(* PLC project Untitled1, Eindhoven University of Technology (TU/e) CIF to Structured Text 0.0 *)
(* stored: creationDateTime 1970-01-01T01:00:00 *)

TYPE STATE : STRUCT
  curTime : LREAL;
  dvar_M_HPC1_HWPump1_ON AT %Q* : BOOL;
  dvar_M_HPC1_HWPump1 AT %Q* : enum_E;
  dvar_M_HPC1_HWPump2_ON AT %Q* : BOOL;
  dvar_M_HPC1_HWPump2 AT %Q* : enum_E;
  dvar_M_HPC1_HWSensorS1 AT %Q* : enum_E;
  dvar_M_HPC1_HWSensorS2 AT %Q* : enum_E;
  dvar_M_HPC1_HWSensorS3 AT %Q* : enum_E;
  dvar_M_HPC1_HWSensorS4 AT %Q* : enum_E;
  dvar_M_HPC1_HWSensorS5 AT %Q* : enum_E;
  dvar_M_HWHPC1ControlButtonAuto_StopLoop AT %Q* : BOOL;
  dvar_M_HWHPC1ControlButtonAuto AT %Q* : enum_E;
  dvar_M_HWHPC1ControlButtonManual_StopLoop AT %Q* : BOOL;
  dvar_M_HWHPC1ControlButtonManual AT %Q* : enum_E;
  dvar_M_HWHPC1ControlMode_AUTO AT %Q* : BOOL;
  dvar_M_HWHPC1ControlMode AT %Q* : enum_E;
  dvar_M_HWHPC1Mode_DRAIN AT %Q* : BOOL;
  dvar_M_HWHPC1Mode_STORE AT %Q* : BOOL;
  dvar_M_HWHPC1Mode_OFF AT %Q* : BOOL;
  dvar_M_HWHPC1Mode AT %Q* : enum_E;
  dvar_M_HWHPC1ModeButtonDrain_StopLoop AT %Q* : BOOL;
  dvar_M_HWHPC1ModeButtonDrain AT %Q* : enum_E;
  dvar_M_HWHPC1ModeButtonOff_StopLoop AT %Q* : BOOL;
  dvar_M_HWHPC1ModeButtonOff AT %Q* : enum_E;
  dvar_M_HWHPC1ModeButtonStore_StopLoop AT %Q* : BOOL;
  dvar_M_HWHPC1ModeButtonStore AT %Q* : enum_E;
  dvar_M_HWModeTraffictube1Observer AT %Q* : enum_E;
  dvar_M_HWModeTraffictube2Observer AT %Q* : enum_E;
  dvar_M_HWMPCControlButtonAuto_StopLoop AT %Q* : BOOL;
  dvar_M_HWMPCControlButtonAuto AT %Q* : enum_E;
  dvar_M_HWMPCControlButtonManual_StopLoop AT %Q* : BOOL;
  dvar_M_HWMPCControlButtonManual AT %Q* : enum_E;
  dvar_M_HWMPCControlMode_AUTO AT %Q* : BOOL;
  dvar_M_HWMPCControlMode AT %Q* : enum_E;
  dvar_M_HWMPCMode_DRAIN AT %Q* : BOOL;
  dvar_M_HWMPCMode_STORE AT %Q* : BOOL;
  dvar_M_HWMPCMode_OFF AT %Q* : BOOL;
  dvar_M_HWMPCMode AT %Q* : enum_E;
  dvar_M_HWMPCModeButtonDrain_StopLoop AT %Q* : BOOL;
  dvar_M_HWMPCModeButtonDrain AT %Q* : enum_E;
  dvar_M_HWMPCModeButtonOff_StopLoop AT %Q* : BOOL;
  dvar_M_HWMPCModeButtonOff AT %Q* : enum_E;
  dvar_M_HWMPCModeButtonStore_StopLoop AT %Q* : BOOL;
  dvar_M_HWMPCModeButtonStore AT %Q* : enum_E;
  dvar_M_HWMutex1_Here AT %Q* : BOOL;
  dvar_M_HWMutex1_SendingAway AT %Q* : BOOL;
  dvar_M_HWMutex1 AT %Q* : enum_E;
  dvar_M_HWMutex2_Here AT %Q* : BOOL;
  dvar_M_HWMutex2_SendingAway AT %Q* : BOOL;
  dvar_M_HWMutex2 AT %Q* : enum_E;
  dvar_M_HWMutex3_Here AT %Q* : BOOL;
  dvar_M_HWMutex3_SendingAway AT %Q* : BOOL;
  dvar_M_HWMutex3 AT %Q* : enum_E;
  dvar_M_HWMutex4_Here AT %Q* : BOOL;
  dvar_M_HWMutex4_SendingAway AT %Q* : BOOL;
  dvar_M_HWMutex4 AT %Q* : enum_E;
  dvar_M_MPC_HWPomprichting_HPC1 AT %Q* : BOOL;
  dvar_M_MPC_HWPomprichting AT %Q* : enum_E;
  dvar_M_MPC_HWPump1_ON AT %Q* : BOOL;
  dvar_M_MPC_HWPump1 AT %Q* : enum_E;
  dvar_M_MPC_HWPump2_ON AT %Q* : BOOL;
  dvar_M_MPC_HWPump2 AT %Q* : enum_E;
  dvar_M_MPC_HWSensorS1 AT %Q* : enum_E;
  dvar_M_MPC_HWSensorS2 AT %Q* : enum_E;
  dvar_M_MPC_HWSensorS3 AT %Q* : enum_E;
  dvar_M_MPC_HWSensorS4 AT %Q* : enum_E;
  dvar_M_MPC_HWSensorS5 AT %Q* : enum_E;
  dvar_M_Mutex1Home_TokenTracker AT %Q* : enum_E;
  dvar_M_Mutex2Home_TokenTracker AT %Q* : enum_E;
  dvar_M_Mutex3Home_TokenTracker AT %Q* : enum_E;
  dvar_M_Mutex4Home_TokenTracker AT %Q* : enum_E;
  dvar_M_Pumpcellars_HeadPumpcellar1_Control_ButtonAuto AT %Q* : enum_E;
  dvar_M_Pumpcellars_HeadPumpcellar1_Control_ButtonDrain AT %Q* : enum_E;
  dvar_M_Pumpcellars_HeadPumpcellar1_Control_ButtonManual AT %Q* : enum_E;
  dvar_M_Pumpcellars_HeadPumpcellar1_Control_ButtonOff AT %Q* : enum_E;
  dvar_M_Pumpcellars_HeadPumpcellar1_Control_ButtonStore AT %Q* : enum_E;
  dvar_M_Pumpcellars_HeadPumpcellar1_Control_Mode AT %Q* : enum_E;
  dvar_M_Pumpcellars_HeadPumpcellar1_Control_Observer AT %Q* : enum_E;
  dvar_M_Pumpcellars_HeadPumpcellar1_Mode AT %Q* : enum_E;
  dvar_M_Pumpcellars_HeadPumpcellar1_Pump1 AT %Q* : enum_E;
  dvar_M_Pumpcellars_HeadPumpcellar1_Pump2 AT %Q* : enum_E;
  dvar_M_Pumpcellars_HeadPumpcellar1_SensorTank AT %Q* : enum_E;
  dvar_M_Pumpcellars_MiddlePumpcellar_Control_ButtonAuto AT %Q* : enum_E;
  dvar_M_Pumpcellars_MiddlePumpcellar_Control_ButtonDrain AT %Q* : enum_E;
  dvar_M_Pumpcellars_MiddlePumpcellar_Control_ButtonManual AT %Q* : enum_E;
  dvar_M_Pumpcellars_MiddlePumpcellar_Control_ButtonOff AT %Q* : enum_E;
  dvar_M_Pumpcellars_MiddlePumpcellar_Control_ButtonStore AT %Q* : enum_E;
  dvar_M_Pumpcellars_MiddlePumpcellar_Control_Mode AT %Q* : enum_E;
  dvar_M_Pumpcellars_MiddlePumpcellar_Control_Observer AT %Q* : enum_E;
  dvar_M_Pumpcellars_MiddlePumpcellar_Mode AT %Q* : enum_E;
  dvar_M_Pumpcellars_MiddlePumpcellar_Pump1 AT %Q* : enum_E;
  dvar_M_Pumpcellars_MiddlePumpcellar_Pump2 AT %Q* : enum_E;
  dvar_M_Pumpcellars_MiddlePumpcellar_PumpDirection AT %Q* : enum_E;
  dvar_M_Pumpcellars_MiddlePumpcellar_SensorTank AT %Q* : enum_E;
  dvar_M_Pumpcellars_Traffictube1_ModeTraffictube_Observer AT %Q* : enum_E;
  dvar_M_Pumpcellars_Traffictube2_ModeTraffictube_Observer AT %Q* : enum_E;
  dvar_M_RequirementStateEvtExcls AT %Q* : enum_E;
  dvar_M_sup1a AT %Q* : enum_E;
  dvar_M_sup2 AT %Q* : enum_E;
  dvar_M_sup4 AT %Q* : enum_E;
  dvar_M_sup5 AT %Q* : enum_E;
  dvar_M_sup8 AT %Q* : enum_E;
END_STRUCT;
END_TYPE

TYPE enum_E : (elit_auto, elit_autoPressed, elit_Away, elit_drain, elit_drainPressed, elit_emergency, elit_Empty, elit_headPumpcellar1, elit_headPumpcellar2, elit_Home, elit_IdleHere, elit_IdleNotHere, elit_manual, elit_manualPressed, elit_off, elit_offPressed, elit_on, elit_operational, elit_recovery, elit_S1, elit_S2, elit_S3, elit_S4, elit_S5, elit_Sending, elit_store, elit_storePressed, elit_unpressed, elit_X);
END_TYPE

FUNCTION alg_MPCStoreAllowed : BOOL
  VAR_INPUT
    state : STATE;
  END_VAR

            alg_MPCStoreAllowed := ((((state.dvar_M_Pumpcellars_MiddlePumpcellar_Control_Observer) = (elit_unpressed)) OR (((state.dvar_M_Pumpcellars_MiddlePumpcellar_Control_Mode) = (elit_manual)) AND ((state.dvar_M_Pumpcellars_MiddlePumpcellar_Control_Observer) <> (elit_autoPressed)))) AND ((((state.dvar_M_Pumpcellars_MiddlePumpcellar_Control_Mode) = (elit_auto)) AND (NOT(((state.dvar_M_Pumpcellars_Traffictube1_ModeTraffictube_Observer) = (elit_operational)) AND ((state.dvar_M_Pumpcellars_Traffictube2_ModeTraffictube_Observer) = (elit_operational))))) OR (((state.dvar_M_Pumpcellars_MiddlePumpcellar_Control_Mode) = (elit_manual)) AND ((state.dvar_M_Pumpcellars_MiddlePumpcellar_Control_Observer) = (elit_storePressed))))) AND (((state.dvar_M_Pumpcellars_MiddlePumpcellar_Mode) = (elit_drain)) OR ((state.dvar_M_Pumpcellars_MiddlePumpcellar_Mode) = (elit_off)));
          
END_FUNCTION

FUNCTION alg_MPCDrainAllowed : BOOL
  VAR_INPUT
    state : STATE;
  END_VAR

            alg_MPCDrainAllowed := ((((state.dvar_M_Pumpcellars_MiddlePumpcellar_Control_Observer) = (elit_unpressed)) OR (((state.dvar_M_Pumpcellars_MiddlePumpcellar_Control_Mode) = (elit_manual)) AND ((state.dvar_M_Pumpcellars_MiddlePumpcellar_Control_Observer) <> (elit_autoPressed)))) AND ((((state.dvar_M_Pumpcellars_MiddlePumpcellar_Control_Mode) = (elit_auto)) AND (((state.dvar_M_Pumpcellars_Traffictube1_ModeTraffictube_Observer) = (elit_operational)) AND ((state.dvar_M_Pumpcellars_Traffictube2_ModeTraffictube_Observer) = (elit_operational)))) OR (((state.dvar_M_Pumpcellars_MiddlePumpcellar_Control_Mode) = (elit_manual)) AND ((state.dvar_M_Pumpcellars_MiddlePumpcellar_Control_Observer) = (elit_drainPressed))))) AND (((state.dvar_M_Pumpcellars_MiddlePumpcellar_Mode) = (elit_store)) OR ((state.dvar_M_Pumpcellars_MiddlePumpcellar_Mode) = (elit_off)));
          
END_FUNCTION

FUNCTION alg_MPCOffAllowed : BOOL
  VAR_INPUT
    state : STATE;
  END_VAR

            alg_MPCOffAllowed := ((((state.dvar_M_Pumpcellars_MiddlePumpcellar_Control_Observer) = (elit_unpressed)) OR (((state.dvar_M_Pumpcellars_MiddlePumpcellar_Control_Mode) = (elit_manual)) AND ((state.dvar_M_Pumpcellars_MiddlePumpcellar_Control_Observer) <> (elit_autoPressed)))) AND (((state.dvar_M_Pumpcellars_MiddlePumpcellar_Control_Mode) = (elit_manual)) AND ((state.dvar_M_Pumpcellars_MiddlePumpcellar_Control_Observer) = (elit_offPressed)))) AND (((state.dvar_M_Pumpcellars_MiddlePumpcellar_Mode) = (elit_drain)) OR ((state.dvar_M_Pumpcellars_MiddlePumpcellar_Mode) = (elit_store)));
          
END_FUNCTION

FUNCTION alg_HPC1StoreAllowed : BOOL
  VAR_INPUT
    state : STATE;
  END_VAR

            alg_HPC1StoreAllowed := ((((state.dvar_M_Pumpcellars_HeadPumpcellar1_Control_Observer) = (elit_unpressed)) OR (((state.dvar_M_Pumpcellars_HeadPumpcellar1_Control_Mode) = (elit_manual)) AND ((state.dvar_M_Pumpcellars_HeadPumpcellar1_Control_Observer) <> (elit_autoPressed)))) AND ((((state.dvar_M_Pumpcellars_HeadPumpcellar1_Control_Mode) = (elit_auto)) AND (NOT(((state.dvar_M_Pumpcellars_Traffictube1_ModeTraffictube_Observer) = (elit_operational)) AND ((state.dvar_M_Pumpcellars_Traffictube2_ModeTraffictube_Observer) = (elit_operational))))) OR (((state.dvar_M_Pumpcellars_HeadPumpcellar1_Control_Mode) = (elit_manual)) AND ((state.dvar_M_Pumpcellars_HeadPumpcellar1_Control_Observer) = (elit_storePressed))))) AND (((state.dvar_M_Pumpcellars_HeadPumpcellar1_Mode) = (elit_drain)) OR ((state.dvar_M_Pumpcellars_HeadPumpcellar1_Mode) = (elit_off)));
          
END_FUNCTION

FUNCTION alg_HPC1DrainAllowed : BOOL
  VAR_INPUT
    state : STATE;
  END_VAR

            alg_HPC1DrainAllowed := ((((state.dvar_M_Pumpcellars_HeadPumpcellar1_Control_Observer) = (elit_unpressed)) OR (((state.dvar_M_Pumpcellars_HeadPumpcellar1_Control_Mode) = (elit_manual)) AND ((state.dvar_M_Pumpcellars_HeadPumpcellar1_Control_Observer) <> (elit_autoPressed)))) AND ((((state.dvar_M_Pumpcellars_HeadPumpcellar1_Control_Mode) = (elit_auto)) AND (((state.dvar_M_Pumpcellars_Traffictube1_ModeTraffictube_Observer) = (elit_operational)) AND ((state.dvar_M_Pumpcellars_Traffictube2_ModeTraffictube_Observer) = (elit_operational)))) OR (((state.dvar_M_Pumpcellars_HeadPumpcellar1_Control_Mode) = (elit_manual)) AND ((state.dvar_M_Pumpcellars_HeadPumpcellar1_Control_Observer) = (elit_drainPressed))))) AND (((state.dvar_M_Pumpcellars_HeadPumpcellar1_Mode) = (elit_store)) OR ((state.dvar_M_Pumpcellars_HeadPumpcellar1_Mode) = (elit_off)));
          
END_FUNCTION

FUNCTION alg_HPC1OffAllowed : BOOL
  VAR_INPUT
    state : STATE;
  END_VAR

            alg_HPC1OffAllowed := ((((state.dvar_M_Pumpcellars_HeadPumpcellar1_Control_Observer) = (elit_unpressed)) OR (((state.dvar_M_Pumpcellars_HeadPumpcellar1_Control_Mode) = (elit_manual)) AND ((state.dvar_M_Pumpcellars_HeadPumpcellar1_Control_Observer) <> (elit_autoPressed)))) AND (((state.dvar_M_Pumpcellars_HeadPumpcellar1_Control_Mode) = (elit_manual)) AND ((state.dvar_M_Pumpcellars_HeadPumpcellar1_Control_Observer) = (elit_offPressed)))) AND (((state.dvar_M_Pumpcellars_HeadPumpcellar1_Mode) = (elit_drain)) OR ((state.dvar_M_Pumpcellars_HeadPumpcellar1_Mode) = (elit_store)));
          
END_FUNCTION

FUNCTION alg_Mutex1HomeReturnCondition : BOOL
  VAR_INPUT
    state : STATE;
  END_VAR

            alg_Mutex1HomeReturnCondition := ((NOT(alg_MPCStoreAllowed(state))) AND (NOT(alg_MPCDrainAllowed(state)))) AND (NOT(alg_MPCOffAllowed(state)));
          
END_FUNCTION

FUNCTION alg_Mutex2HomeReturnCondition : BOOL
  VAR_INPUT
    state : STATE;
  END_VAR

            alg_Mutex2HomeReturnCondition := ((NOT(alg_MPCStoreAllowed(state))) AND (NOT(alg_MPCDrainAllowed(state)))) AND (NOT(alg_MPCOffAllowed(state)));
          
END_FUNCTION

FUNCTION alg_Mutex3HomeReturnCondition : BOOL
  VAR_INPUT
    state : STATE;
  END_VAR

            alg_Mutex3HomeReturnCondition := ((NOT(alg_HPC1StoreAllowed(state))) AND (NOT(alg_HPC1DrainAllowed(state)))) AND (NOT(alg_HPC1OffAllowed(state)));
          
END_FUNCTION

FUNCTION alg_Mutex4HomeReturnCondition : BOOL
  VAR_INPUT
    state : STATE;
  END_VAR

            alg_Mutex4HomeReturnCondition := ((NOT(alg_HPC1StoreAllowed(state))) AND (NOT(alg_HPC1DrainAllowed(state)))) AND (NOT(alg_HPC1OffAllowed(state)));
          
END_FUNCTION

FUNCTION alg_Mutex1Home_ReturnCondition : BOOL
  VAR_INPUT
    state : STATE;
  END_VAR

            alg_Mutex1Home_ReturnCondition := alg_Mutex1HomeReturnCondition(state);
          
END_FUNCTION

FUNCTION alg_Mutex2Home_ReturnCondition : BOOL
  VAR_INPUT
    state : STATE;
  END_VAR

            alg_Mutex2Home_ReturnCondition := alg_Mutex2HomeReturnCondition(state);
          
END_FUNCTION

FUNCTION alg_Mutex3Home_ReturnCondition : BOOL
  VAR_INPUT
    state : STATE;
  END_VAR

            alg_Mutex3Home_ReturnCondition := alg_Mutex3HomeReturnCondition(state);
          
END_FUNCTION

FUNCTION alg_Mutex4Home_ReturnCondition : BOOL
  VAR_INPUT
    state : STATE;
  END_VAR

            alg_Mutex4Home_ReturnCondition := alg_Mutex4HomeReturnCondition(state);
          
END_FUNCTION

FUNCTION alg_M_HWMutex1_InitiallyHere : BOOL
  VAR_INPUT
    state : STATE;
  END_VAR

            alg_M_HWMutex1_InitiallyHere := TRUE;
          
END_FUNCTION

FUNCTION alg_M_HWMutex2_InitiallyHere : BOOL
  VAR_INPUT
    state : STATE;
  END_VAR

            alg_M_HWMutex2_InitiallyHere := TRUE;
          
END_FUNCTION

FUNCTION alg_M_HWMutex3_InitiallyHere : BOOL
  VAR_INPUT
    state : STATE;
  END_VAR

            alg_M_HWMutex3_InitiallyHere := TRUE;
          
END_FUNCTION

FUNCTION alg_M_HWMutex4_InitiallyHere : BOOL
  VAR_INPUT
    state : STATE;
  END_VAR

            alg_M_HWMutex4_InitiallyHere := TRUE;
          
END_FUNCTION

PROGRAM MAIN
  VAR_OUTPUT
    timerValue0 : TIME;
    timerValue1 : TIME;
  END_VAR
  VAR
    cnt : LINT;
    first : BOOL := TRUE;
    curTimerValue : TIME;
    state0 : STATE;
    curTime : LREAL;
    loopsKilled : LINT;
  END_VAR
  VAR_TEMP
    lastTimerValue : TIME;
    curDeltaTime : TIME;
    curDeltaSecs : LREAL;
    state1 : STATE;
    progress : BOOL;
    loopCount : INT;
    b1 : BOOL;
    b2 : BOOL;
    b3 : BOOL;
    b4 : BOOL;
    b5 : BOOL;
  END_VAR

            
// Handle 'time' and cycle time.
cnt := cnt + 1;

timer0(IN := curTimer = 0, PT := T#1D);
timer1(IN := curTimer = 1, PT := T#1D);
timerValue0 := timer0.ET;
timerValue1 := timer1.ET;

lastTimerValue := curTimerValue;
IF curTimer = 0 THEN
    curTimerValue := timerValue0;
ELSE
    curTimerValue := timerValue1;
END_IF;
curDeltaTime := curTimerValue - lastTimerValue;
curDeltaSecs := TIME_TO_LREAL(curDeltaTime) / 1000;
curTime := curTime + curDeltaSecs;

IF cnt MOD 10 = 0 THEN
    curTimer := 1 - curTimer;
    curTimerValue := T#0S;
    timer0(IN := curTimer = 0, PT := T#1D);
    timer1(IN := curTimer = 1, PT := T#1D);
    timerValue0 := timer0.ET;
    timerValue1 := timer1.ET;
END_IF;

IF first THEN
    first := FALSE;

    // Initialize state variables for initial state.
    state0.dvar_M_HPC1_HWPump1_ON := FALSE;
    state0.dvar_M_HPC1_HWPump1 := elit_X;
    state0.dvar_M_HPC1_HWPump2_ON := FALSE;
    state0.dvar_M_HPC1_HWPump2 := elit_X;
    state0.dvar_M_HPC1_HWSensorS1 := elit_off;
    state0.dvar_M_HPC1_HWSensorS2 := elit_off;
    state0.dvar_M_HPC1_HWSensorS3 := elit_off;
    state0.dvar_M_HPC1_HWSensorS4 := elit_off;
    state0.dvar_M_HPC1_HWSensorS5 := elit_off;
    state0.dvar_M_HWHPC1ControlButtonAuto_StopLoop := FALSE;
    state0.dvar_M_HWHPC1ControlButtonAuto := elit_X;
    state0.dvar_M_HWHPC1ControlButtonManual_StopLoop := FALSE;
    state0.dvar_M_HWHPC1ControlButtonManual := elit_X;
    state0.dvar_M_HWHPC1ControlMode_AUTO := TRUE;
    state0.dvar_M_HWHPC1ControlMode := elit_X;
    state0.dvar_M_HWHPC1Mode_DRAIN := TRUE;
    state0.dvar_M_HWHPC1Mode_STORE := FALSE;
    state0.dvar_M_HWHPC1Mode_OFF := FALSE;
    state0.dvar_M_HWHPC1Mode := elit_drain;
    state0.dvar_M_HWHPC1ModeButtonDrain_StopLoop := FALSE;
    state0.dvar_M_HWHPC1ModeButtonDrain := elit_X;
    state0.dvar_M_HWHPC1ModeButtonOff_StopLoop := FALSE;
    state0.dvar_M_HWHPC1ModeButtonOff := elit_X;
    state0.dvar_M_HWHPC1ModeButtonStore_StopLoop := FALSE;
    state0.dvar_M_HWHPC1ModeButtonStore := elit_X;
    state0.dvar_M_HWModeTraffictube1Observer := elit_X;
    state0.dvar_M_HWModeTraffictube2Observer := elit_X;
    state0.dvar_M_HWMPCControlButtonAuto_StopLoop := FALSE;
    state0.dvar_M_HWMPCControlButtonAuto := elit_X;
    state0.dvar_M_HWMPCControlButtonManual_StopLoop := FALSE;
    state0.dvar_M_HWMPCControlButtonManual := elit_X;
    state0.dvar_M_HWMPCControlMode_AUTO := TRUE;
    state0.dvar_M_HWMPCControlMode := elit_X;
    state0.dvar_M_HWMPCMode_DRAIN := TRUE;
    state0.dvar_M_HWMPCMode_STORE := FALSE;
    state0.dvar_M_HWMPCMode_OFF := FALSE;
    state0.dvar_M_HWMPCMode := elit_drain;
    state0.dvar_M_HWMPCModeButtonDrain_StopLoop := FALSE;
    state0.dvar_M_HWMPCModeButtonDrain := elit_X;
    state0.dvar_M_HWMPCModeButtonOff_StopLoop := FALSE;
    state0.dvar_M_HWMPCModeButtonOff := elit_X;
    state0.dvar_M_HWMPCModeButtonStore_StopLoop := FALSE;
    state0.dvar_M_HWMPCModeButtonStore := elit_X;
    state0.dvar_M_HWMutex1_Here := TRUE;
    state0.dvar_M_HWMutex1_SendingAway := FALSE;
    state0.dvar_M_HWMutex1 := elit_IdleHere;
    state0.dvar_M_HWMutex2_Here := TRUE;
    state0.dvar_M_HWMutex2_SendingAway := FALSE;
    state0.dvar_M_HWMutex2 := elit_IdleHere;
    state0.dvar_M_HWMutex3_Here := TRUE;
    state0.dvar_M_HWMutex3_SendingAway := FALSE;
    state0.dvar_M_HWMutex3 := elit_IdleHere;
    state0.dvar_M_HWMutex4_Here := TRUE;
    state0.dvar_M_HWMutex4_SendingAway := FALSE;
    state0.dvar_M_HWMutex4 := elit_IdleHere;
    state0.dvar_M_MPC_HWPomprichting_HPC1 := TRUE;
    state0.dvar_M_MPC_HWPomprichting := elit_X;
    state0.dvar_M_MPC_HWPump1_ON := FALSE;
    state0.dvar_M_MPC_HWPump1 := elit_X;
    state0.dvar_M_MPC_HWPump2_ON := FALSE;
    state0.dvar_M_MPC_HWPump2 := elit_X;
    state0.dvar_M_MPC_HWSensorS1 := elit_off;
    state0.dvar_M_MPC_HWSensorS2 := elit_off;
    state0.dvar_M_MPC_HWSensorS3 := elit_off;
    state0.dvar_M_MPC_HWSensorS4 := elit_off;
    state0.dvar_M_MPC_HWSensorS5 := elit_off;
    state0.dvar_M_Mutex1Home_TokenTracker := elit_Home;
    state0.dvar_M_Mutex2Home_TokenTracker := elit_Home;
    state0.dvar_M_Mutex3Home_TokenTracker := elit_Home;
    state0.dvar_M_Mutex4Home_TokenTracker := elit_Home;
    state0.dvar_M_Pumpcellars_HeadPumpcellar1_Control_ButtonAuto := elit_X;
    state0.dvar_M_Pumpcellars_HeadPumpcellar1_Control_ButtonDrain := elit_X;
    state0.dvar_M_Pumpcellars_HeadPumpcellar1_Control_ButtonManual := elit_X;
    state0.dvar_M_Pumpcellars_HeadPumpcellar1_Control_ButtonOff := elit_X;
    state0.dvar_M_Pumpcellars_HeadPumpcellar1_Control_ButtonStore := elit_X;
    state0.dvar_M_Pumpcellars_HeadPumpcellar1_Control_Mode := elit_auto;
    state0.dvar_M_Pumpcellars_HeadPumpcellar1_Control_Observer := elit_unpressed;
    state0.dvar_M_Pumpcellars_HeadPumpcellar1_Mode := elit_drain;
    state0.dvar_M_Pumpcellars_HeadPumpcellar1_Pump1 := elit_off;
    state0.dvar_M_Pumpcellars_HeadPumpcellar1_Pump2 := elit_off;
    state0.dvar_M_Pumpcellars_HeadPumpcellar1_SensorTank := elit_Empty;
    state0.dvar_M_Pumpcellars_MiddlePumpcellar_Control_ButtonAuto := elit_X;
    state0.dvar_M_Pumpcellars_MiddlePumpcellar_Control_ButtonDrain := elit_X;
    state0.dvar_M_Pumpcellars_MiddlePumpcellar_Control_ButtonManual := elit_X;
    state0.dvar_M_Pumpcellars_MiddlePumpcellar_Control_ButtonOff := elit_X;
    state0.dvar_M_Pumpcellars_MiddlePumpcellar_Control_ButtonStore := elit_X;
    state0.dvar_M_Pumpcellars_MiddlePumpcellar_Control_Mode := elit_auto;
    state0.dvar_M_Pumpcellars_MiddlePumpcellar_Control_Observer := elit_unpressed;
    state0.dvar_M_Pumpcellars_MiddlePumpcellar_Mode := elit_drain;
    state0.dvar_M_Pumpcellars_MiddlePumpcellar_Pump1 := elit_off;
    state0.dvar_M_Pumpcellars_MiddlePumpcellar_Pump2 := elit_off;
    state0.dvar_M_Pumpcellars_MiddlePumpcellar_PumpDirection := elit_headPumpcellar1;
    state0.dvar_M_Pumpcellars_MiddlePumpcellar_SensorTank := elit_Empty;
    state0.dvar_M_Pumpcellars_Traffictube1_ModeTraffictube_Observer := elit_operational;
    state0.dvar_M_Pumpcellars_Traffictube2_ModeTraffictube_Observer := elit_operational;
    state0.dvar_M_RequirementStateEvtExcls := elit_X;
    state0.dvar_M_sup1a := elit_X;
    state0.dvar_M_sup2 := elit_X;
    state0.dvar_M_sup4 := elit_X;
    state0.dvar_M_sup5 := elit_X;
    state0.dvar_M_sup8 := elit_X;
ELSE
    // Update continuous variables for time delay.

    state0.curTime := curTime;
END_IF;

// Event loop.
WHILE TRUE DO
    progress := FALSE;

    // Event "M.HWMutex1_c_finishSending".
    IF NOT progress THEN
        b1 := (state0.dvar_M_HWMutex1) = (elit_Sending);
        b1 := b1 AND (ivar_M_HWMutex1_There);
        IF b1 THEN
            progress := TRUE;
            state1 := state0;

            state1.dvar_M_HWMutex1_SendingAway := FALSE;
            state1.dvar_M_HWMutex1 := elit_IdleNotHere;

            state0 := state1;
        END_IF;
    END_IF;

    // Event "M.HWMutex2_c_finishSending".
    IF NOT progress THEN
        b1 := (state0.dvar_M_HWMutex2) = (elit_Sending);
        b1 := b1 AND (ivar_M_HWMutex2_There);
        IF b1 THEN
            progress := TRUE;
            state1 := state0;

            state1.dvar_M_HWMutex2_SendingAway := FALSE;
            state1.dvar_M_HWMutex2 := elit_IdleNotHere;

            state0 := state1;
        END_IF;
    END_IF;

    // Event "M.HWMutex3_c_finishSending".
    IF NOT progress THEN
        b1 := (state0.dvar_M_HWMutex3) = (elit_Sending);
        b1 := b1 AND (ivar_M_HWMutex3_There);
        IF b1 THEN
            progress := TRUE;
            state1 := state0;

            state1.dvar_M_HWMutex3_SendingAway := FALSE;
            state1.dvar_M_HWMutex3 := elit_IdleNotHere;

            state0 := state1;
        END_IF;
    END_IF;

    // Event "M.HWMutex4_c_finishSending".
    IF NOT progress THEN
        b1 := (state0.dvar_M_HWMutex4) = (elit_Sending);
        b1 := b1 AND (ivar_M_HWMutex4_There);
        IF b1 THEN
            progress := TRUE;
            state1 := state0;

            state1.dvar_M_HWMutex4_SendingAway := FALSE;
            state1.dvar_M_HWMutex4 := elit_IdleNotHere;

            state0 := state1;
        END_IF;
    END_IF;

    // Event "Mutex1Home_TokenTracker_c_receive".
    IF NOT progress THEN
        b1 := (state0.dvar_M_HWMutex1) = (elit_IdleNotHere);
        b1 := b1 AND (ivar_M_HWMutex1_SendingHere);
        b1 := b1 AND ((state0.dvar_M_Mutex1Home_TokenTracker) = (elit_Away));
        IF b1 THEN
            progress := TRUE;
            state1 := state0;

            state1.dvar_M_HWMutex1_Here := TRUE;
            state1.dvar_M_HWMutex1 := elit_IdleHere;
            state1.dvar_M_Mutex1Home_TokenTracker := elit_Home;

            state0 := state1;
        END_IF;
    END_IF;

    // Event "Mutex1Home_TokenTracker_c_send".
    IF NOT progress THEN
        b1 := (state0.dvar_M_HWMutex1) = (elit_IdleHere);
        b1 := b1 AND ((ivar_M_HWMutex1_SendingHere) = (FALSE));
        b1 := b1 AND (state0.dvar_M_HWMutex1_Here);
        b1 := b1 AND ((state0.dvar_M_Mutex1Home_TokenTracker) = (elit_Home));
        b1 := b1 AND ((state0.dvar_M_RequirementStateEvtExcls) = (elit_X));
        b1 := b1 AND (alg_Mutex1Home_ReturnCondition(state0));
        b1 := b1 AND (ivar_Mutex1Home_R2);
        IF b1 THEN
            progress := TRUE;
            state1 := state0;

            state1.dvar_M_HWMutex1_SendingAway := TRUE;
            state1.dvar_M_HWMutex1_Here := FALSE;
            state1.dvar_M_HWMutex1 := elit_Sending;
            state1.dvar_M_Mutex1Home_TokenTracker := elit_Away;

            state0 := state1;
        END_IF;
    END_IF;

    // Event "Mutex2Home_TokenTracker_c_receive".
    IF NOT progress THEN
        b1 := (state0.dvar_M_HWMutex2) = (elit_IdleNotHere);
        b1 := b1 AND (ivar_M_HWMutex2_SendingHere);
        b1 := b1 AND ((state0.dvar_M_Mutex2Home_TokenTracker) = (elit_Away));
        IF b1 THEN
            progress := TRUE;
            state1 := state0;

            state1.dvar_M_HWMutex2_Here := TRUE;
            state1.dvar_M_HWMutex2 := elit_IdleHere;
            state1.dvar_M_Mutex2Home_TokenTracker := elit_Home;

            state0 := state1;
        END_IF;
    END_IF;

    // Event "Mutex2Home_TokenTracker_c_send".
    IF NOT progress THEN
        b1 := (state0.dvar_M_HWMutex2) = (elit_IdleHere);
        b1 := b1 AND ((ivar_M_HWMutex2_SendingHere) = (FALSE));
        b1 := b1 AND (state0.dvar_M_HWMutex2_Here);
        b1 := b1 AND ((state0.dvar_M_Mutex2Home_TokenTracker) = (elit_Home));
        b1 := b1 AND ((state0.dvar_M_RequirementStateEvtExcls) = (elit_X));
        b1 := b1 AND (alg_Mutex2Home_ReturnCondition(state0));
        b1 := b1 AND (ivar_Mutex2Home_R2);
        IF b1 THEN
            progress := TRUE;
            state1 := state0;

            state1.dvar_M_HWMutex2_SendingAway := TRUE;
            state1.dvar_M_HWMutex2_Here := FALSE;
            state1.dvar_M_HWMutex2 := elit_Sending;
            state1.dvar_M_Mutex2Home_TokenTracker := elit_Away;

            state0 := state1;
        END_IF;
    END_IF;

    // Event "Mutex3Home_TokenTracker_c_receive".
    IF NOT progress THEN
        b1 := (state0.dvar_M_HWMutex3) = (elit_IdleNotHere);
        b1 := b1 AND (ivar_M_HWMutex3_SendingHere);
        b1 := b1 AND ((state0.dvar_M_Mutex3Home_TokenTracker) = (elit_Away));
        IF b1 THEN
            progress := TRUE;
            state1 := state0;

            state1.dvar_M_HWMutex3_Here := TRUE;
            state1.dvar_M_HWMutex3 := elit_IdleHere;
            state1.dvar_M_Mutex3Home_TokenTracker := elit_Home;

            state0 := state1;
        END_IF;
    END_IF;

    // Event "Mutex3Home_TokenTracker_c_send".
    IF NOT progress THEN
        b1 := (state0.dvar_M_HWMutex3) = (elit_IdleHere);
        b1 := b1 AND ((ivar_M_HWMutex3_SendingHere) = (FALSE));
        b1 := b1 AND (state0.dvar_M_HWMutex3_Here);
        b1 := b1 AND ((state0.dvar_M_Mutex3Home_TokenTracker) = (elit_Home));
        b1 := b1 AND ((state0.dvar_M_RequirementStateEvtExcls) = (elit_X));
        b1 := b1 AND (alg_Mutex3Home_ReturnCondition(state0));
        b1 := b1 AND (ivar_Mutex3Home_R2);
        IF b1 THEN
            progress := TRUE;
            state1 := state0;

            state1.dvar_M_HWMutex3_SendingAway := TRUE;
            state1.dvar_M_HWMutex3_Here := FALSE;
            state1.dvar_M_HWMutex3 := elit_Sending;
            state1.dvar_M_Mutex3Home_TokenTracker := elit_Away;

            state0 := state1;
        END_IF;
    END_IF;

    // Event "Mutex4Home_TokenTracker_c_receive".
    IF NOT progress THEN
        b1 := (state0.dvar_M_HWMutex4) = (elit_IdleNotHere);
        b1 := b1 AND (ivar_M_HWMutex4_SendingHere);
        b1 := b1 AND ((state0.dvar_M_Mutex4Home_TokenTracker) = (elit_Away));
        IF b1 THEN
            progress := TRUE;
            state1 := state0;

            state1.dvar_M_HWMutex4_Here := TRUE;
            state1.dvar_M_HWMutex4 := elit_IdleHere;
            state1.dvar_M_Mutex4Home_TokenTracker := elit_Home;

            state0 := state1;
        END_IF;
    END_IF;

    // Event "Mutex4Home_TokenTracker_c_send".
    IF NOT progress THEN
        b1 := (state0.dvar_M_HWMutex4) = (elit_IdleHere);
        b1 := b1 AND ((ivar_M_HWMutex4_SendingHere) = (FALSE));
        b1 := b1 AND (state0.dvar_M_HWMutex4_Here);
        b1 := b1 AND ((state0.dvar_M_Mutex4Home_TokenTracker) = (elit_Home));
        b1 := b1 AND ((state0.dvar_M_RequirementStateEvtExcls) = (elit_X));
        b1 := b1 AND (alg_Mutex4Home_ReturnCondition(state0));
        b1 := b1 AND (ivar_Mutex4Home_R2);
        IF b1 THEN
            progress := TRUE;
            state1 := state0;

            state1.dvar_M_HWMutex4_SendingAway := TRUE;
            state1.dvar_M_HWMutex4_Here := FALSE;
            state1.dvar_M_HWMutex4 := elit_Sending;
            state1.dvar_M_Mutex4Home_TokenTracker := elit_Away;

            state0 := state1;
        END_IF;
    END_IF;

    // Event "Pumpcellars_HeadPumpcellar1_Control_ButtonAuto_u_push".
    IF NOT progress THEN
        b1 := (state0.dvar_M_HWHPC1ControlButtonAuto) = (elit_X);
        b1 := b1 AND (ivar_M_HWHPC1ControlButtonAuto_PUSHED);
        b1 := b1 AND (NOT(state0.dvar_M_HWHPC1ControlButtonAuto_StopLoop));
        b1 := b1 AND ((state0.dvar_M_Pumpcellars_HeadPumpcellar1_Control_ButtonAuto) = (elit_X));
        IF b1 THEN
            b3 := (state0.dvar_M_Pumpcellars_HeadPumpcellar1_Control_Observer) = (elit_unpressed);
            IF b3 THEN
                b4 := (state0.dvar_M_Pumpcellars_HeadPumpcellar1_Control_Mode) = (elit_manual);
                b4 := b4 OR ((state0.dvar_M_Pumpcellars_HeadPumpcellar1_Control_Mode) <> (elit_manual));
                b3 := b3 AND (b4);
            END_IF;
            b2 := b3;
            b2 := b2 OR ((state0.dvar_M_Pumpcellars_HeadPumpcellar1_Control_Observer) = (elit_autoPressed));
            b2 := b2 OR ((state0.dvar_M_Pumpcellars_HeadPumpcellar1_Control_Observer) = (elit_manualPressed));
            b2 := b2 OR ((state0.dvar_M_Pumpcellars_HeadPumpcellar1_Control_Observer) = (elit_storePressed));
            b2 := b2 OR ((state0.dvar_M_Pumpcellars_HeadPumpcellar1_Control_Observer) = (elit_drainPressed));
            b2 := b2 OR ((state0.dvar_M_Pumpcellars_HeadPumpcellar1_Control_Observer) = (elit_offPressed));
            b1 := b1 AND (b2);
        END_IF;
        IF b1 THEN
            progress := TRUE;
            state1 := state0;

            state1.dvar_M_HWHPC1ControlButtonAuto_StopLoop := TRUE;
            IF (((state0.dvar_M_Pumpcellars_HeadPumpcellar1_Control_Observer) = (elit_unpressed)) AND ((state0.dvar_M_Pumpcellars_HeadPumpcellar1_Control_Mode) = (elit_manual))) THEN
                state1.dvar_M_Pumpcellars_HeadPumpcellar1_Control_Observer := elit_autoPressed;
            ELSIF (((state0.dvar_M_Pumpcellars_HeadPumpcellar1_Control_Observer) = (elit_unpressed)) AND ((state0.dvar_M_Pumpcellars_HeadPumpcellar1_Control_Mode) <> (elit_manual))) THEN
                state1.dvar_M_Pumpcellars_HeadPumpcellar1_Control_Observer := elit_unpressed;
            ELSIF ((state0.dvar_M_Pumpcellars_HeadPumpcellar1_Control_Observer) = (elit_autoPressed)) THEN
                state1.dvar_M_Pumpcellars_HeadPumpcellar1_Control_Observer := elit_autoPressed;
            ELSIF ((state0.dvar_M_Pumpcellars_HeadPumpcellar1_Control_Observer) = (elit_manualPressed)) THEN
                state1.dvar_M_Pumpcellars_HeadPumpcellar1_Control_Observer := elit_manualPressed;
            ELSIF ((state0.dvar_M_Pumpcellars_HeadPumpcellar1_Control_Observer) = (elit_storePressed)) THEN
                state1.dvar_M_Pumpcellars_HeadPumpcellar1_Control_Observer := elit_storePressed;
            ELSIF ((state0.dvar_M_Pumpcellars_HeadPumpcellar1_Control_Observer) = (elit_drainPressed)) THEN
                state1.dvar_M_Pumpcellars_HeadPumpcellar1_Control_Observer := elit_drainPressed;
            ELSIF ((state0.dvar_M_Pumpcellars_HeadPumpcellar1_Control_Observer) = (elit_offPressed)) THEN
                state1.dvar_M_Pumpcellars_HeadPumpcellar1_Control_Observer := elit_offPressed;
            END_IF;

            state0 := state1;
        END_IF;
    END_IF;

    // Event "Pumpcellars_HeadPumpcellar1_Control_ButtonDrain_u_push".
    IF NOT progress THEN
        b1 := (state0.dvar_M_HWHPC1ModeButtonDrain) = (elit_X);
        b1 := b1 AND (ivar_M_HWHPC1ModeButtonDrain_PUSHED);
        b1 := b1 AND (NOT(state0.dvar_M_HWHPC1ModeButtonDrain_StopLoop));
        b1 := b1 AND ((state0.dvar_M_Pumpcellars_HeadPumpcellar1_Control_ButtonDrain) = (elit_X));
        IF b1 THEN
            b3 := (state0.dvar_M_Pumpcellars_HeadPumpcellar1_Control_Observer) = (elit_unpressed);
            IF b3 THEN
                b5 := (state0.dvar_M_Pumpcellars_HeadPumpcellar1_Control_Mode) = (elit_manual);
                b5 := b5 AND ((state0.dvar_M_Pumpcellars_HeadPumpcellar1_Mode) <> (elit_drain));
                b4 := b5;
                b4 := b4 OR (NOT(((state0.dvar_M_Pumpcellars_HeadPumpcellar1_Control_Mode) = (elit_manual)) AND ((state0.dvar_M_Pumpcellars_HeadPumpcellar1_Mode) <> (elit_drain))));
                b3 := b3 AND (b4);
            END_IF;
            b2 := b3;
            b2 := b2 OR ((state0.dvar_M_Pumpcellars_HeadPumpcellar1_Control_Observer) = (elit_autoPressed));
            b2 := b2 OR ((state0.dvar_M_Pumpcellars_HeadPumpcellar1_Control_Observer) = (elit_manualPressed));
            b2 := b2 OR ((state0.dvar_M_Pumpcellars_HeadPumpcellar1_Control_Observer) = (elit_storePressed));
            b2 := b2 OR ((state0.dvar_M_Pumpcellars_HeadPumpcellar1_Control_Observer) = (elit_drainPressed));
            b2 := b2 OR ((state0.dvar_M_Pumpcellars_HeadPumpcellar1_Control_Observer) = (elit_offPressed));
            b1 := b1 AND (b2);
        END_IF;
        IF b1 THEN
            progress := TRUE;
            state1 := state0;

            state1.dvar_M_HWHPC1ModeButtonDrain_StopLoop := TRUE;
            IF (((state0.dvar_M_Pumpcellars_HeadPumpcellar1_Control_Observer) = (elit_unpressed)) AND (((state0.dvar_M_Pumpcellars_HeadPumpcellar1_Control_Mode) = (elit_manual)) AND ((state0.dvar_M_Pumpcellars_HeadPumpcellar1_Mode) <> (elit_drain)))) THEN
                state1.dvar_M_Pumpcellars_HeadPumpcellar1_Control_Observer := elit_drainPressed;
            ELSIF (((state0.dvar_M_Pumpcellars_HeadPumpcellar1_Control_Observer) = (elit_unpressed)) AND (NOT(((state0.dvar_M_Pumpcellars_HeadPumpcellar1_Control_Mode) = (elit_manual)) AND ((state0.dvar_M_Pumpcellars_HeadPumpcellar1_Mode) <> (elit_drain))))) THEN
                state1.dvar_M_Pumpcellars_HeadPumpcellar1_Control_Observer := elit_unpressed;
            ELSIF ((state0.dvar_M_Pumpcellars_HeadPumpcellar1_Control_Observer) = (elit_autoPressed)) THEN
                state1.dvar_M_Pumpcellars_HeadPumpcellar1_Control_Observer := elit_autoPressed;
            ELSIF ((state0.dvar_M_Pumpcellars_HeadPumpcellar1_Control_Observer) = (elit_manualPressed)) THEN
                state1.dvar_M_Pumpcellars_HeadPumpcellar1_Control_Observer := elit_manualPressed;
            ELSIF ((state0.dvar_M_Pumpcellars_HeadPumpcellar1_Control_Observer) = (elit_storePressed)) THEN
                state1.dvar_M_Pumpcellars_HeadPumpcellar1_Control_Observer := elit_storePressed;
            ELSIF ((state0.dvar_M_Pumpcellars_HeadPumpcellar1_Control_Observer) = (elit_drainPressed)) THEN
                state1.dvar_M_Pumpcellars_HeadPumpcellar1_Control_Observer := elit_drainPressed;
            ELSIF ((state0.dvar_M_Pumpcellars_HeadPumpcellar1_Control_Observer) = (elit_offPressed)) THEN
                state1.dvar_M_Pumpcellars_HeadPumpcellar1_Control_Observer := elit_offPressed;
            END_IF;

            state0 := state1;
        END_IF;
    END_IF;

    // Event "Pumpcellars_HeadPumpcellar1_Control_ButtonManual_u_push".
    IF NOT progress THEN
        b1 := (state0.dvar_M_HWHPC1ControlButtonManual) = (elit_X);
        b1 := b1 AND (ivar_M_HWHPC1ControlButtonManual_PUSHED);
        b1 := b1 AND (NOT(state0.dvar_M_HWHPC1ControlButtonManual_StopLoop));
        b1 := b1 AND ((state0.dvar_M_Pumpcellars_HeadPumpcellar1_Control_ButtonManual) = (elit_X));
        IF b1 THEN
            b3 := (state0.dvar_M_Pumpcellars_HeadPumpcellar1_Control_Observer) = (elit_unpressed);
            IF b3 THEN
                b4 := (state0.dvar_M_Pumpcellars_HeadPumpcellar1_Control_Mode) = (elit_auto);
                b4 := b4 OR ((state0.dvar_M_Pumpcellars_HeadPumpcellar1_Control_Mode) <> (elit_auto));
                b3 := b3 AND (b4);
            END_IF;
            b2 := b3;
            b2 := b2 OR ((state0.dvar_M_Pumpcellars_HeadPumpcellar1_Control_Observer) = (elit_autoPressed));
            b2 := b2 OR ((state0.dvar_M_Pumpcellars_HeadPumpcellar1_Control_Observer) = (elit_manualPressed));
            b2 := b2 OR ((state0.dvar_M_Pumpcellars_HeadPumpcellar1_Control_Observer) = (elit_storePressed));
            b2 := b2 OR ((state0.dvar_M_Pumpcellars_HeadPumpcellar1_Control_Observer) = (elit_drainPressed));
            b2 := b2 OR ((state0.dvar_M_Pumpcellars_HeadPumpcellar1_Control_Observer) = (elit_offPressed));
            b1 := b1 AND (b2);
        END_IF;
        IF b1 THEN
            progress := TRUE;
            state1 := state0;

            state1.dvar_M_HWHPC1ControlButtonManual_StopLoop := TRUE;
            IF (((state0.dvar_M_Pumpcellars_HeadPumpcellar1_Control_Observer) = (elit_unpressed)) AND ((state0.dvar_M_Pumpcellars_HeadPumpcellar1_Control_Mode) = (elit_auto))) THEN
                state1.dvar_M_Pumpcellars_HeadPumpcellar1_Control_Observer := elit_manualPressed;
            ELSIF (((state0.dvar_M_Pumpcellars_HeadPumpcellar1_Control_Observer) = (elit_unpressed)) AND ((state0.dvar_M_Pumpcellars_HeadPumpcellar1_Control_Mode) <> (elit_auto))) THEN
                state1.dvar_M_Pumpcellars_HeadPumpcellar1_Control_Observer := elit_unpressed;
            ELSIF ((state0.dvar_M_Pumpcellars_HeadPumpcellar1_Control_Observer) = (elit_autoPressed)) THEN
                state1.dvar_M_Pumpcellars_HeadPumpcellar1_Control_Observer := elit_autoPressed;
            ELSIF ((state0.dvar_M_Pumpcellars_HeadPumpcellar1_Control_Observer) = (elit_manualPressed)) THEN
                state1.dvar_M_Pumpcellars_HeadPumpcellar1_Control_Observer := elit_manualPressed;
            ELSIF ((state0.dvar_M_Pumpcellars_HeadPumpcellar1_Control_Observer) = (elit_storePressed)) THEN
                state1.dvar_M_Pumpcellars_HeadPumpcellar1_Control_Observer := elit_storePressed;
            ELSIF ((state0.dvar_M_Pumpcellars_HeadPumpcellar1_Control_Observer) = (elit_drainPressed)) THEN
                state1.dvar_M_Pumpcellars_HeadPumpcellar1_Control_Observer := elit_drainPressed;
            ELSIF ((state0.dvar_M_Pumpcellars_HeadPumpcellar1_Control_Observer) = (elit_offPressed)) THEN
                state1.dvar_M_Pumpcellars_HeadPumpcellar1_Control_Observer := elit_offPressed;
            END_IF;

            state0 := state1;
        END_IF;
    END_IF;

    // Event "Pumpcellars_HeadPumpcellar1_Control_ButtonOff_u_push".
    IF NOT progress THEN
        b1 := (state0.dvar_M_HWHPC1ModeButtonOff) = (elit_X);
        b1 := b1 AND (ivar_M_HWHPC1ModeButtonOff_PUSHED);
        b1 := b1 AND (NOT(state0.dvar_M_HWHPC1ModeButtonOff_StopLoop));
        b1 := b1 AND ((state0.dvar_M_Pumpcellars_HeadPumpcellar1_Control_ButtonOff) = (elit_X));
        IF b1 THEN
            b3 := (state0.dvar_M_Pumpcellars_HeadPumpcellar1_Control_Observer) = (elit_unpressed);
            IF b3 THEN
                b5 := (state0.dvar_M_Pumpcellars_HeadPumpcellar1_Control_Mode) = (elit_manual);
                b5 := b5 AND ((state0.dvar_M_Pumpcellars_HeadPumpcellar1_Mode) <> (elit_off));
                b4 := b5;
                b4 := b4 OR (NOT(((state0.dvar_M_Pumpcellars_HeadPumpcellar1_Control_Mode) = (elit_manual)) AND ((state0.dvar_M_Pumpcellars_HeadPumpcellar1_Mode) <> (elit_off))));
                b3 := b3 AND (b4);
            END_IF;
            b2 := b3;
            b2 := b2 OR ((state0.dvar_M_Pumpcellars_HeadPumpcellar1_Control_Observer) = (elit_autoPressed));
            b2 := b2 OR ((state0.dvar_M_Pumpcellars_HeadPumpcellar1_Control_Observer) = (elit_manualPressed));
            b2 := b2 OR ((state0.dvar_M_Pumpcellars_HeadPumpcellar1_Control_Observer) = (elit_storePressed));
            b2 := b2 OR ((state0.dvar_M_Pumpcellars_HeadPumpcellar1_Control_Observer) = (elit_drainPressed));
            b2 := b2 OR ((state0.dvar_M_Pumpcellars_HeadPumpcellar1_Control_Observer) = (elit_offPressed));
            b1 := b1 AND (b2);
        END_IF;
        IF b1 THEN
            progress := TRUE;
            state1 := state0;

            state1.dvar_M_HWHPC1ModeButtonOff_StopLoop := TRUE;
            IF (((state0.dvar_M_Pumpcellars_HeadPumpcellar1_Control_Observer) = (elit_unpressed)) AND (((state0.dvar_M_Pumpcellars_HeadPumpcellar1_Control_Mode) = (elit_manual)) AND ((state0.dvar_M_Pumpcellars_HeadPumpcellar1_Mode) <> (elit_off)))) THEN
                state1.dvar_M_Pumpcellars_HeadPumpcellar1_Control_Observer := elit_offPressed;
            ELSIF (((state0.dvar_M_Pumpcellars_HeadPumpcellar1_Control_Observer) = (elit_unpressed)) AND (NOT(((state0.dvar_M_Pumpcellars_HeadPumpcellar1_Control_Mode) = (elit_manual)) AND ((state0.dvar_M_Pumpcellars_HeadPumpcellar1_Mode) <> (elit_off))))) THEN
                state1.dvar_M_Pumpcellars_HeadPumpcellar1_Control_Observer := elit_unpressed;
            ELSIF ((state0.dvar_M_Pumpcellars_HeadPumpcellar1_Control_Observer) = (elit_autoPressed)) THEN
                state1.dvar_M_Pumpcellars_HeadPumpcellar1_Control_Observer := elit_autoPressed;
            ELSIF ((state0.dvar_M_Pumpcellars_HeadPumpcellar1_Control_Observer) = (elit_manualPressed)) THEN
                state1.dvar_M_Pumpcellars_HeadPumpcellar1_Control_Observer := elit_manualPressed;
            ELSIF ((state0.dvar_M_Pumpcellars_HeadPumpcellar1_Control_Observer) = (elit_storePressed)) THEN
                state1.dvar_M_Pumpcellars_HeadPumpcellar1_Control_Observer := elit_storePressed;
            ELSIF ((state0.dvar_M_Pumpcellars_HeadPumpcellar1_Control_Observer) = (elit_drainPressed)) THEN
                state1.dvar_M_Pumpcellars_HeadPumpcellar1_Control_Observer := elit_drainPressed;
            ELSIF ((state0.dvar_M_Pumpcellars_HeadPumpcellar1_Control_Observer) = (elit_offPressed)) THEN
                state1.dvar_M_Pumpcellars_HeadPumpcellar1_Control_Observer := elit_offPressed;
            END_IF;

            state0 := state1;
        END_IF;
    END_IF;

    // Event "Pumpcellars_HeadPumpcellar1_Control_ButtonStore_u_push".
    IF NOT progress THEN
        b1 := (state0.dvar_M_HWHPC1ModeButtonStore) = (elit_X);
        b1 := b1 AND (ivar_M_HWHPC1ModeButtonStore_PUSHED);
        b1 := b1 AND (NOT(state0.dvar_M_HWHPC1ModeButtonStore_StopLoop));
        b1 := b1 AND ((state0.dvar_M_Pumpcellars_HeadPumpcellar1_Control_ButtonStore) = (elit_X));
        IF b1 THEN
            b3 := (state0.dvar_M_Pumpcellars_HeadPumpcellar1_Control_Observer) = (elit_unpressed);
            IF b3 THEN
                b5 := (state0.dvar_M_Pumpcellars_HeadPumpcellar1_Control_Mode) = (elit_manual);
                b5 := b5 AND ((state0.dvar_M_Pumpcellars_HeadPumpcellar1_Mode) <> (elit_store));
                b4 := b5;
                b4 := b4 OR (NOT(((state0.dvar_M_Pumpcellars_HeadPumpcellar1_Control_Mode) = (elit_manual)) AND ((state0.dvar_M_Pumpcellars_HeadPumpcellar1_Mode) <> (elit_store))));
                b3 := b3 AND (b4);
            END_IF;
            b2 := b3;
            b2 := b2 OR ((state0.dvar_M_Pumpcellars_HeadPumpcellar1_Control_Observer) = (elit_autoPressed));
            b2 := b2 OR ((state0.dvar_M_Pumpcellars_HeadPumpcellar1_Control_Observer) = (elit_manualPressed));
            b2 := b2 OR ((state0.dvar_M_Pumpcellars_HeadPumpcellar1_Control_Observer) = (elit_storePressed));
            b2 := b2 OR ((state0.dvar_M_Pumpcellars_HeadPumpcellar1_Control_Observer) = (elit_drainPressed));
            b2 := b2 OR ((state0.dvar_M_Pumpcellars_HeadPumpcellar1_Control_Observer) = (elit_offPressed));
            b1 := b1 AND (b2);
        END_IF;
        IF b1 THEN
            progress := TRUE;
            state1 := state0;

            state1.dvar_M_HWHPC1ModeButtonStore_StopLoop := TRUE;
            IF (((state0.dvar_M_Pumpcellars_HeadPumpcellar1_Control_Observer) = (elit_unpressed)) AND (((state0.dvar_M_Pumpcellars_HeadPumpcellar1_Control_Mode) = (elit_manual)) AND ((state0.dvar_M_Pumpcellars_HeadPumpcellar1_Mode) <> (elit_store)))) THEN
                state1.dvar_M_Pumpcellars_HeadPumpcellar1_Control_Observer := elit_storePressed;
            ELSIF (((state0.dvar_M_Pumpcellars_HeadPumpcellar1_Control_Observer) = (elit_unpressed)) AND (NOT(((state0.dvar_M_Pumpcellars_HeadPumpcellar1_Control_Mode) = (elit_manual)) AND ((state0.dvar_M_Pumpcellars_HeadPumpcellar1_Mode) <> (elit_store))))) THEN
                state1.dvar_M_Pumpcellars_HeadPumpcellar1_Control_Observer := elit_unpressed;
            ELSIF ((state0.dvar_M_Pumpcellars_HeadPumpcellar1_Control_Observer) = (elit_autoPressed)) THEN
                state1.dvar_M_Pumpcellars_HeadPumpcellar1_Control_Observer := elit_autoPressed;
            ELSIF ((state0.dvar_M_Pumpcellars_HeadPumpcellar1_Control_Observer) = (elit_manualPressed)) THEN
                state1.dvar_M_Pumpcellars_HeadPumpcellar1_Control_Observer := elit_manualPressed;
            ELSIF ((state0.dvar_M_Pumpcellars_HeadPumpcellar1_Control_Observer) = (elit_storePressed)) THEN
                state1.dvar_M_Pumpcellars_HeadPumpcellar1_Control_Observer := elit_storePressed;
            ELSIF ((state0.dvar_M_Pumpcellars_HeadPumpcellar1_Control_Observer) = (elit_drainPressed)) THEN
                state1.dvar_M_Pumpcellars_HeadPumpcellar1_Control_Observer := elit_drainPressed;
            ELSIF ((state0.dvar_M_Pumpcellars_HeadPumpcellar1_Control_Observer) = (elit_offPressed)) THEN
                state1.dvar_M_Pumpcellars_HeadPumpcellar1_Control_Observer := elit_offPressed;
            END_IF;

            state0 := state1;
        END_IF;
    END_IF;

    // Event "Pumpcellars_HeadPumpcellar1_Control_Mode_c_auto".
    IF NOT progress THEN
        b1 := (state0.dvar_M_HWHPC1ControlMode) = (elit_X);
        b1 := b1 AND ((state0.dvar_M_Pumpcellars_HeadPumpcellar1_Control_Mode) = (elit_manual));
        b1 := b1 AND ((state0.dvar_M_RequirementStateEvtExcls) = (elit_X));
        b1 := b1 AND ((state0.dvar_M_Pumpcellars_HeadPumpcellar1_Control_Observer) = (elit_autoPressed));
        b1 := b1 AND ((state0.dvar_M_sup1a) = (elit_X));
        b1 := b1 AND ((state0.dvar_M_sup5) = (elit_X));
        b1 := b1 AND ((state0.dvar_M_sup8) = (elit_X));
        IF b1 THEN
            progress := TRUE;
            state1 := state0;

            state1.dvar_M_HWHPC1ControlMode_AUTO := TRUE;
            state1.dvar_M_Pumpcellars_HeadPumpcellar1_Control_Mode := elit_auto;

            state0 := state1;
        END_IF;
    END_IF;

    // Event "Pumpcellars_HeadPumpcellar1_Control_Mode_c_manual".
    IF NOT progress THEN
        b1 := (state0.dvar_M_HWHPC1ControlMode) = (elit_X);
        b1 := b1 AND ((state0.dvar_M_Pumpcellars_HeadPumpcellar1_Control_Mode) = (elit_auto));
        b1 := b1 AND ((state0.dvar_M_RequirementStateEvtExcls) = (elit_X));
        b1 := b1 AND ((state0.dvar_M_Pumpcellars_HeadPumpcellar1_Control_Observer) = (elit_manualPressed));
        b1 := b1 AND ((state0.dvar_M_sup1a) = (elit_X));
        b1 := b1 AND ((state0.dvar_M_sup5) = (elit_X));
        b1 := b1 AND ((state0.dvar_M_sup8) = (elit_X));
        IF b1 THEN
            progress := TRUE;
            state1 := state0;

            state1.dvar_M_HWHPC1ControlMode_AUTO := FALSE;
            state1.dvar_M_Pumpcellars_HeadPumpcellar1_Control_Mode := elit_manual;

            state0 := state1;
        END_IF;
    END_IF;

    // Event "Pumpcellars_HeadPumpcellar1_Control_Observer_c_done".
    IF NOT progress THEN
        b1 := (state0.dvar_M_HWHPC1ControlButtonAuto) = (elit_X);
        b1 := b1 AND ((state0.dvar_M_HWHPC1ControlButtonManual) = (elit_X));
        b1 := b1 AND ((state0.dvar_M_HWHPC1ModeButtonDrain) = (elit_X));
        b1 := b1 AND ((state0.dvar_M_HWHPC1ModeButtonOff) = (elit_X));
        b1 := b1 AND ((state0.dvar_M_HWHPC1ModeButtonStore) = (elit_X));
        IF b1 THEN
            b3 := (state0.dvar_M_Pumpcellars_HeadPumpcellar1_Control_Observer) = (elit_autoPressed);
            b3 := b3 AND ((state0.dvar_M_Pumpcellars_HeadPumpcellar1_Control_Mode) = (elit_auto));
            b2 := b3;
            IF NOT(b2) THEN
                b3 := (state0.dvar_M_Pumpcellars_HeadPumpcellar1_Control_Observer) = (elit_manualPressed);
                b3 := b3 AND ((state0.dvar_M_Pumpcellars_HeadPumpcellar1_Control_Mode) = (elit_manual));
                b2 := b2 OR (b3);
            END_IF;
            IF NOT(b2) THEN
                b3 := (state0.dvar_M_Pumpcellars_HeadPumpcellar1_Control_Observer) = (elit_storePressed);
                b3 := b3 AND ((state0.dvar_M_Pumpcellars_HeadPumpcellar1_Mode) = (elit_store));
                b2 := b2 OR (b3);
            END_IF;
            IF NOT(b2) THEN
                b3 := (state0.dvar_M_Pumpcellars_HeadPumpcellar1_Control_Observer) = (elit_drainPressed);
                b3 := b3 AND ((state0.dvar_M_Pumpcellars_HeadPumpcellar1_Mode) = (elit_drain));
                b2 := b2 OR (b3);
            END_IF;
            IF NOT(b2) THEN
                b3 := (state0.dvar_M_Pumpcellars_HeadPumpcellar1_Control_Observer) = (elit_offPressed);
                b3 := b3 AND ((state0.dvar_M_Pumpcellars_HeadPumpcellar1_Mode) = (elit_off));
                b2 := b2 OR (b3);
            END_IF;
            b1 := b1 AND (b2);
        END_IF;
        b1 := b1 AND ((state0.dvar_M_sup1a) = (elit_X));
        b1 := b1 AND ((state0.dvar_M_sup5) = (elit_X));
        b1 := b1 AND ((state0.dvar_M_sup8) = (elit_X));
        IF b1 THEN
            progress := TRUE;
            state1 := state0;

            state1.dvar_M_HWHPC1ControlButtonAuto_StopLoop := FALSE;
            state1.dvar_M_HWHPC1ControlButtonManual_StopLoop := FALSE;
            state1.dvar_M_HWHPC1ModeButtonDrain_StopLoop := FALSE;
            state1.dvar_M_HWHPC1ModeButtonOff_StopLoop := FALSE;
            state1.dvar_M_HWHPC1ModeButtonStore_StopLoop := FALSE;
            IF (((state0.dvar_M_Pumpcellars_HeadPumpcellar1_Control_Observer) = (elit_autoPressed)) AND ((state0.dvar_M_Pumpcellars_HeadPumpcellar1_Control_Mode) = (elit_auto))) THEN
                state1.dvar_M_Pumpcellars_HeadPumpcellar1_Control_Observer := elit_unpressed;
            ELSIF (((state0.dvar_M_Pumpcellars_HeadPumpcellar1_Control_Observer) = (elit_manualPressed)) AND ((state0.dvar_M_Pumpcellars_HeadPumpcellar1_Control_Mode) = (elit_manual))) THEN
                state1.dvar_M_Pumpcellars_HeadPumpcellar1_Control_Observer := elit_unpressed;
            ELSIF (((state0.dvar_M_Pumpcellars_HeadPumpcellar1_Control_Observer) = (elit_storePressed)) AND ((state0.dvar_M_Pumpcellars_HeadPumpcellar1_Mode) = (elit_store))) THEN
                state1.dvar_M_Pumpcellars_HeadPumpcellar1_Control_Observer := elit_unpressed;
            ELSIF (((state0.dvar_M_Pumpcellars_HeadPumpcellar1_Control_Observer) = (elit_drainPressed)) AND ((state0.dvar_M_Pumpcellars_HeadPumpcellar1_Mode) = (elit_drain))) THEN
                state1.dvar_M_Pumpcellars_HeadPumpcellar1_Control_Observer := elit_unpressed;
            ELSIF (((state0.dvar_M_Pumpcellars_HeadPumpcellar1_Control_Observer) = (elit_offPressed)) AND ((state0.dvar_M_Pumpcellars_HeadPumpcellar1_Mode) = (elit_off))) THEN
                state1.dvar_M_Pumpcellars_HeadPumpcellar1_Control_Observer := elit_unpressed;
            END_IF;

            state0 := state1;
        END_IF;
    END_IF;

    // Event "Pumpcellars_HeadPumpcellar1_Mode_c_drain".
    IF NOT progress THEN
        b2 := (state0.dvar_M_Pumpcellars_HeadPumpcellar1_Mode) = (elit_store);
        b2 := b2 OR ((state0.dvar_M_Pumpcellars_HeadPumpcellar1_Mode) = (elit_off));
        b1 := b2;
        b1 := b1 AND ((state0.dvar_M_RequirementStateEvtExcls) = (elit_X));
        IF b1 THEN
            b2 := (state0.dvar_M_Pumpcellars_HeadPumpcellar1_Control_Observer) = (elit_unpressed);
            IF NOT(b2) THEN
                b3 := (state0.dvar_M_Pumpcellars_HeadPumpcellar1_Control_Mode) = (elit_manual);
                b3 := b3 AND ((state0.dvar_M_Pumpcellars_HeadPumpcellar1_Control_Observer) <> (elit_autoPressed));
                b2 := b2 OR (b3);
            END_IF;
            b1 := b1 AND (b2);
        END_IF;
        IF b1 THEN
            b3 := (state0.dvar_M_Pumpcellars_HeadPumpcellar1_Control_Mode) = (elit_auto);
            b3 := b3 AND ((state0.dvar_M_Pumpcellars_Traffictube1_ModeTraffictube_Observer) = (elit_operational));
            b3 := b3 AND ((state0.dvar_M_Pumpcellars_Traffictube2_ModeTraffictube_Observer) = (elit_operational));
            b2 := b3;
            IF NOT(b2) THEN
                b3 := (state0.dvar_M_Pumpcellars_HeadPumpcellar1_Control_Mode) = (elit_manual);
                b3 := b3 AND ((state0.dvar_M_Pumpcellars_HeadPumpcellar1_Control_Observer) = (elit_drainPressed));
                b2 := b2 OR (b3);
            END_IF;
            b1 := b1 AND (b2);
        END_IF;
        b1 := b1 AND ((state0.dvar_M_Mutex3Home_TokenTracker) = (elit_Home));
        b1 := b1 AND ((state0.dvar_M_Mutex4Home_TokenTracker) = (elit_Home));
        b1 := b1 AND ((state0.dvar_M_sup1a) = (elit_X));
        b1 := b1 AND ((state0.dvar_M_sup5) = (elit_X));
        b1 := b1 AND ((state0.dvar_M_sup8) = (elit_X));
        IF b1 THEN
            progress := TRUE;
            state1 := state0;

            IF ((state0.dvar_M_HWHPC1Mode) = (elit_drain)) THEN
                state1.dvar_M_HWHPC1Mode := elit_drain;
            ELSIF ((state0.dvar_M_HWHPC1Mode) = (elit_store)) THEN
                state1.dvar_M_HWHPC1Mode_DRAIN := TRUE;
                state1.dvar_M_HWHPC1Mode_STORE := FALSE;
                state1.dvar_M_HWHPC1Mode_OFF := FALSE;
                state1.dvar_M_HWHPC1Mode := elit_drain;
            ELSIF ((state0.dvar_M_HWHPC1Mode) = (elit_off)) THEN
                state1.dvar_M_HWHPC1Mode_DRAIN := TRUE;
                state1.dvar_M_HWHPC1Mode_STORE := FALSE;
                state1.dvar_M_HWHPC1Mode_OFF := FALSE;
                state1.dvar_M_HWHPC1Mode := elit_drain;
            END_IF;
            IF ((state0.dvar_M_Pumpcellars_HeadPumpcellar1_Mode) = (elit_store)) THEN
                state1.dvar_M_Pumpcellars_HeadPumpcellar1_Mode := elit_drain;
            ELSIF ((state0.dvar_M_Pumpcellars_HeadPumpcellar1_Mode) = (elit_off)) THEN
                state1.dvar_M_Pumpcellars_HeadPumpcellar1_Mode := elit_drain;
            END_IF;

            state0 := state1;
        END_IF;
    END_IF;

    // Event "Pumpcellars_HeadPumpcellar1_Mode_c_off".
    IF NOT progress THEN
        b2 := (state0.dvar_M_Pumpcellars_HeadPumpcellar1_Mode) = (elit_drain);
        b2 := b2 OR ((state0.dvar_M_Pumpcellars_HeadPumpcellar1_Mode) = (elit_store));
        b1 := b2;
        b1 := b1 AND ((state0.dvar_M_RequirementStateEvtExcls) = (elit_X));
        IF b1 THEN
            b2 := (state0.dvar_M_Pumpcellars_HeadPumpcellar1_Control_Observer) = (elit_unpressed);
            IF NOT(b2) THEN
                b3 := (state0.dvar_M_Pumpcellars_HeadPumpcellar1_Control_Mode) = (elit_manual);
                b3 := b3 AND ((state0.dvar_M_Pumpcellars_HeadPumpcellar1_Control_Observer) <> (elit_autoPressed));
                b2 := b2 OR (b3);
            END_IF;
            b1 := b1 AND (b2);
        END_IF;
        b1 := b1 AND ((state0.dvar_M_Pumpcellars_HeadPumpcellar1_Control_Mode) = (elit_manual));
        b1 := b1 AND ((state0.dvar_M_Pumpcellars_HeadPumpcellar1_Control_Observer) = (elit_offPressed));
        b1 := b1 AND ((state0.dvar_M_Mutex3Home_TokenTracker) = (elit_Home));
        b1 := b1 AND ((state0.dvar_M_Mutex4Home_TokenTracker) = (elit_Home));
        b1 := b1 AND ((state0.dvar_M_sup1a) = (elit_X));
        b1 := b1 AND ((state0.dvar_M_sup5) = (elit_X));
        b1 := b1 AND ((state0.dvar_M_sup8) = (elit_X));
        IF b1 THEN
            progress := TRUE;
            state1 := state0;

            IF ((state0.dvar_M_HWHPC1Mode) = (elit_drain)) THEN
                state1.dvar_M_HWHPC1Mode_DRAIN := FALSE;
                state1.dvar_M_HWHPC1Mode_STORE := FALSE;
                state1.dvar_M_HWHPC1Mode_OFF := TRUE;
                state1.dvar_M_HWHPC1Mode := elit_off;
            ELSIF ((state0.dvar_M_HWHPC1Mode) = (elit_store)) THEN
                state1.dvar_M_HWHPC1Mode_DRAIN := FALSE;
                state1.dvar_M_HWHPC1Mode_STORE := FALSE;
                state1.dvar_M_HWHPC1Mode_OFF := TRUE;
                state1.dvar_M_HWHPC1Mode := elit_off;
            ELSIF ((state0.dvar_M_HWHPC1Mode) = (elit_off)) THEN
                state1.dvar_M_HWHPC1Mode := elit_off;
            END_IF;
            IF ((state0.dvar_M_Pumpcellars_HeadPumpcellar1_Mode) = (elit_drain)) THEN
                state1.dvar_M_Pumpcellars_HeadPumpcellar1_Mode := elit_off;
            ELSIF ((state0.dvar_M_Pumpcellars_HeadPumpcellar1_Mode) = (elit_store)) THEN
                state1.dvar_M_Pumpcellars_HeadPumpcellar1_Mode := elit_off;
            END_IF;

            state0 := state1;
        END_IF;
    END_IF;

    // Event "Pumpcellars_HeadPumpcellar1_Mode_c_store".
    IF NOT progress THEN
        b2 := (state0.dvar_M_Pumpcellars_HeadPumpcellar1_Mode) = (elit_drain);
        b2 := b2 OR ((state0.dvar_M_Pumpcellars_HeadPumpcellar1_Mode) = (elit_off));
        b1 := b2;
        b1 := b1 AND ((state0.dvar_M_RequirementStateEvtExcls) = (elit_X));
        IF b1 THEN
            b2 := (state0.dvar_M_Pumpcellars_HeadPumpcellar1_Control_Observer) = (elit_unpressed);
            IF NOT(b2) THEN
                b3 := (state0.dvar_M_Pumpcellars_HeadPumpcellar1_Control_Mode) = (elit_manual);
                b3 := b3 AND ((state0.dvar_M_Pumpcellars_HeadPumpcellar1_Control_Observer) <> (elit_autoPressed));
                b2 := b2 OR (b3);
            END_IF;
            b1 := b1 AND (b2);
        END_IF;
        IF b1 THEN
            b3 := (state0.dvar_M_Pumpcellars_HeadPumpcellar1_Control_Mode) = (elit_auto);
            b3 := b3 AND (NOT(((state0.dvar_M_Pumpcellars_Traffictube1_ModeTraffictube_Observer) = (elit_operational)) AND ((state0.dvar_M_Pumpcellars_Traffictube2_ModeTraffictube_Observer) = (elit_operational))));
            b2 := b3;
            IF NOT(b2) THEN
                b3 := (state0.dvar_M_Pumpcellars_HeadPumpcellar1_Control_Mode) = (elit_manual);
                b3 := b3 AND ((state0.dvar_M_Pumpcellars_HeadPumpcellar1_Control_Observer) = (elit_storePressed));
                b2 := b2 OR (b3);
            END_IF;
            b1 := b1 AND (b2);
        END_IF;
        b1 := b1 AND ((state0.dvar_M_Mutex3Home_TokenTracker) = (elit_Home));
        b1 := b1 AND ((state0.dvar_M_Mutex4Home_TokenTracker) = (elit_Home));
        b1 := b1 AND ((state0.dvar_M_sup1a) = (elit_X));
        b1 := b1 AND ((state0.dvar_M_sup5) = (elit_X));
        b1 := b1 AND ((state0.dvar_M_sup8) = (elit_X));
        IF b1 THEN
            progress := TRUE;
            state1 := state0;

            IF ((state0.dvar_M_HWHPC1Mode) = (elit_drain)) THEN
                state1.dvar_M_HWHPC1Mode_DRAIN := FALSE;
                state1.dvar_M_HWHPC1Mode_STORE := TRUE;
                state1.dvar_M_HWHPC1Mode_OFF := FALSE;
                state1.dvar_M_HWHPC1Mode := elit_store;
            ELSIF ((state0.dvar_M_HWHPC1Mode) = (elit_store)) THEN
                state1.dvar_M_HWHPC1Mode := elit_store;
            ELSIF ((state0.dvar_M_HWHPC1Mode) = (elit_off)) THEN
                state1.dvar_M_HWHPC1Mode_DRAIN := FALSE;
                state1.dvar_M_HWHPC1Mode_STORE := TRUE;
                state1.dvar_M_HWHPC1Mode_OFF := FALSE;
                state1.dvar_M_HWHPC1Mode := elit_store;
            END_IF;
            IF ((state0.dvar_M_Pumpcellars_HeadPumpcellar1_Mode) = (elit_drain)) THEN
                state1.dvar_M_Pumpcellars_HeadPumpcellar1_Mode := elit_store;
            ELSIF ((state0.dvar_M_Pumpcellars_HeadPumpcellar1_Mode) = (elit_off)) THEN
                state1.dvar_M_Pumpcellars_HeadPumpcellar1_Mode := elit_store;
            END_IF;

            state0 := state1;
        END_IF;
    END_IF;

    // Event "Pumpcellars_HeadPumpcellar1_Pump1_c_off".
    IF NOT progress THEN
        b1 := (state0.dvar_M_HPC1_HWPump1) = (elit_X);
        b1 := b1 AND ((state0.dvar_M_Pumpcellars_HeadPumpcellar1_Pump1) = (elit_on));
        b1 := b1 AND ((state0.dvar_M_RequirementStateEvtExcls) = (elit_X));
        IF b1 THEN
            b3 := (state0.dvar_M_Pumpcellars_HeadPumpcellar1_Mode) = (elit_store);
            IF b3 THEN
                b4 := (state0.dvar_M_Pumpcellars_HeadPumpcellar1_SensorTank) = (elit_S2);
                b4 := b4 OR ((state0.dvar_M_Pumpcellars_HeadPumpcellar1_SensorTank) = (elit_S3));
                b4 := b4 OR ((state0.dvar_M_Pumpcellars_HeadPumpcellar1_SensorTank) = (elit_S1));
                b4 := b4 OR ((state0.dvar_M_Pumpcellars_HeadPumpcellar1_SensorTank) = (elit_Empty));
                b3 := b3 AND (b4);
            END_IF;
            b2 := b3;
            IF NOT(b2) THEN
                b3 := (state0.dvar_M_Pumpcellars_HeadPumpcellar1_Mode) = (elit_drain);
                b3 := b3 AND ((state0.dvar_M_Pumpcellars_HeadPumpcellar1_SensorTank) = (elit_Empty));
                b2 := b2 OR (b3);
            END_IF;
            b2 := b2 OR ((state0.dvar_M_Pumpcellars_HeadPumpcellar1_Mode) = (elit_off));
            b1 := b1 AND (b2);
        END_IF;
        b1 := b1 AND ((state0.dvar_M_Pumpcellars_HeadPumpcellar1_Control_Observer) = (elit_unpressed));
        b1 := b1 AND ((state0.dvar_M_sup5) = (elit_X));
        IF b1 THEN
            progress := TRUE;
            state1 := state0;

            state1.dvar_M_HPC1_HWPump1_ON := FALSE;
            state1.dvar_M_Pumpcellars_HeadPumpcellar1_Pump1 := elit_off;

            state0 := state1;
        END_IF;
    END_IF;

    // Event "Pumpcellars_HeadPumpcellar1_Pump1_c_on".
    IF NOT progress THEN
        b1 := (state0.dvar_M_HPC1_HWPump1) = (elit_X);
        b1 := b1 AND ((state0.dvar_M_Pumpcellars_HeadPumpcellar1_Pump1) = (elit_off));
        b1 := b1 AND ((state0.dvar_M_RequirementStateEvtExcls) = (elit_X));
        IF b1 THEN
            b3 := (state0.dvar_M_Pumpcellars_HeadPumpcellar1_Mode) = (elit_store);
            b3 := b3 AND ((state0.dvar_M_Pumpcellars_HeadPumpcellar1_SensorTank) = (elit_S5));
            b2 := b3;
            IF NOT(b2) THEN
                b3 := (state0.dvar_M_Pumpcellars_HeadPumpcellar1_Mode) = (elit_drain);
                IF b3 THEN
                    b4 := (state0.dvar_M_Pumpcellars_HeadPumpcellar1_SensorTank) = (elit_S2);
                    b4 := b4 OR ((state0.dvar_M_Pumpcellars_HeadPumpcellar1_SensorTank) = (elit_S3));
                    b4 := b4 OR ((state0.dvar_M_Pumpcellars_HeadPumpcellar1_SensorTank) = (elit_S4));
                    b4 := b4 OR ((state0.dvar_M_Pumpcellars_HeadPumpcellar1_SensorTank) = (elit_S5));
                    b3 := b3 AND (b4);
                END_IF;
                b2 := b2 OR (b3);
            END_IF;
            b1 := b1 AND (b2);
        END_IF;
        b1 := b1 AND ((state0.dvar_M_Pumpcellars_HeadPumpcellar1_Control_Observer) = (elit_unpressed));
        b1 := b1 AND ((state0.dvar_M_sup5) = (elit_X));
        IF b1 THEN
            progress := TRUE;
            state1 := state0;

            state1.dvar_M_HPC1_HWPump1_ON := TRUE;
            state1.dvar_M_Pumpcellars_HeadPumpcellar1_Pump1 := elit_on;

            state0 := state1;
        END_IF;
    END_IF;

    // Event "Pumpcellars_HeadPumpcellar1_Pump2_c_off".
    IF NOT progress THEN
        b1 := (state0.dvar_M_HPC1_HWPump2) = (elit_X);
        b1 := b1 AND ((state0.dvar_M_Pumpcellars_HeadPumpcellar1_Pump2) = (elit_on));
        b1 := b1 AND ((state0.dvar_M_RequirementStateEvtExcls) = (elit_X));
        IF b1 THEN
            b3 := (state0.dvar_M_Pumpcellars_HeadPumpcellar1_Mode) = (elit_store);
            IF b3 THEN
                b4 := (state0.dvar_M_Pumpcellars_HeadPumpcellar1_SensorTank) = (elit_S2);
                b4 := b4 OR ((state0.dvar_M_Pumpcellars_HeadPumpcellar1_SensorTank) = (elit_S3));
                b4 := b4 OR ((state0.dvar_M_Pumpcellars_HeadPumpcellar1_SensorTank) = (elit_S1));
                b4 := b4 OR ((state0.dvar_M_Pumpcellars_HeadPumpcellar1_SensorTank) = (elit_Empty));
                b3 := b3 AND (b4);
            END_IF;
            b2 := b3;
            IF NOT(b2) THEN
                b3 := (state0.dvar_M_Pumpcellars_HeadPumpcellar1_Mode) = (elit_drain);
                b3 := b3 AND ((state0.dvar_M_Pumpcellars_HeadPumpcellar1_SensorTank) = (elit_Empty));
                b2 := b2 OR (b3);
            END_IF;
            b2 := b2 OR ((state0.dvar_M_Pumpcellars_HeadPumpcellar1_Mode) = (elit_off));
            b1 := b1 AND (b2);
        END_IF;
        b1 := b1 AND ((state0.dvar_M_Pumpcellars_HeadPumpcellar1_Control_Observer) = (elit_unpressed));
        b1 := b1 AND ((state0.dvar_M_sup5) = (elit_X));
        IF b1 THEN
            progress := TRUE;
            state1 := state0;

            state1.dvar_M_HPC1_HWPump2_ON := FALSE;
            state1.dvar_M_Pumpcellars_HeadPumpcellar1_Pump2 := elit_off;

            state0 := state1;
        END_IF;
    END_IF;

    // Event "Pumpcellars_HeadPumpcellar1_Pump2_c_on".
    IF NOT progress THEN
        b1 := (state0.dvar_M_HPC1_HWPump2) = (elit_X);
        b1 := b1 AND ((state0.dvar_M_Pumpcellars_HeadPumpcellar1_Pump2) = (elit_off));
        b1 := b1 AND ((state0.dvar_M_RequirementStateEvtExcls) = (elit_X));
        IF b1 THEN
            b3 := (state0.dvar_M_Pumpcellars_HeadPumpcellar1_Mode) = (elit_store);
            b3 := b3 AND ((state0.dvar_M_Pumpcellars_HeadPumpcellar1_SensorTank) = (elit_S5));
            b2 := b3;
            IF NOT(b2) THEN
                b3 := (state0.dvar_M_Pumpcellars_HeadPumpcellar1_Mode) = (elit_drain);
                IF b3 THEN
                    b4 := (state0.dvar_M_Pumpcellars_HeadPumpcellar1_SensorTank) = (elit_S3);
                    b4 := b4 OR ((state0.dvar_M_Pumpcellars_HeadPumpcellar1_SensorTank) = (elit_S4));
                    b4 := b4 OR ((state0.dvar_M_Pumpcellars_HeadPumpcellar1_SensorTank) = (elit_S5));
                    b3 := b3 AND (b4);
                END_IF;
                b2 := b2 OR (b3);
            END_IF;
            b1 := b1 AND (b2);
        END_IF;
        b1 := b1 AND ((state0.dvar_M_Pumpcellars_HeadPumpcellar1_Control_Observer) = (elit_unpressed));
        b1 := b1 AND ((state0.dvar_M_sup5) = (elit_X));
        IF b1 THEN
            progress := TRUE;
            state1 := state0;

            state1.dvar_M_HPC1_HWPump2_ON := TRUE;
            state1.dvar_M_Pumpcellars_HeadPumpcellar1_Pump2 := elit_on;

            state0 := state1;
        END_IF;
    END_IF;

    // Event "Pumpcellars_HeadPumpcellar1_SensorTank_u_S1off".
    IF NOT progress THEN
        b1 := (state0.dvar_M_HPC1_HWSensorS1) = (elit_on);
        b1 := b1 AND (NOT(ivar_M_HPC1_HWSensorS1_ON));
        b1 := b1 AND ((state0.dvar_M_Pumpcellars_HeadPumpcellar1_SensorTank) = (elit_S1));
        IF b1 THEN
            b2 := (state0.dvar_M_Pumpcellars_HeadPumpcellar1_Pump1) = (elit_on);
            b2 := b2 OR ((state0.dvar_M_Pumpcellars_HeadPumpcellar1_Pump2) = (elit_on));
            b1 := b1 AND (b2);
        END_IF;
        IF b1 THEN
            progress := TRUE;
            state1 := state0;

            state1.dvar_M_HPC1_HWSensorS1 := elit_off;
            state1.dvar_M_Pumpcellars_HeadPumpcellar1_SensorTank := elit_Empty;

            state0 := state1;
        END_IF;
    END_IF;

    // Event "Pumpcellars_HeadPumpcellar1_SensorTank_u_S1on".
    IF NOT progress THEN
        b1 := (state0.dvar_M_HPC1_HWSensorS1) = (elit_off);
        b1 := b1 AND (ivar_M_HPC1_HWSensorS1_ON);
        b1 := b1 AND ((state0.dvar_M_Pumpcellars_HeadPumpcellar1_SensorTank) = (elit_Empty));
        IF b1 THEN
            progress := TRUE;
            state1 := state0;

            state1.dvar_M_HPC1_HWSensorS1 := elit_on;
            state1.dvar_M_Pumpcellars_HeadPumpcellar1_SensorTank := elit_S1;

            state0 := state1;
        END_IF;
    END_IF;

    // Event "Pumpcellars_HeadPumpcellar1_SensorTank_u_S2off".
    IF NOT progress THEN
        b1 := (state0.dvar_M_HPC1_HWSensorS2) = (elit_on);
        b1 := b1 AND (NOT(ivar_M_HPC1_HWSensorS2_ON));
        b1 := b1 AND ((state0.dvar_M_Pumpcellars_HeadPumpcellar1_SensorTank) = (elit_S2));
        IF b1 THEN
            b2 := (state0.dvar_M_Pumpcellars_HeadPumpcellar1_Pump1) = (elit_on);
            b2 := b2 OR ((state0.dvar_M_Pumpcellars_HeadPumpcellar1_Pump2) = (elit_on));
            b1 := b1 AND (b2);
        END_IF;
        IF b1 THEN
            progress := TRUE;
            state1 := state0;

            state1.dvar_M_HPC1_HWSensorS2 := elit_off;
            state1.dvar_M_Pumpcellars_HeadPumpcellar1_SensorTank := elit_S1;

            state0 := state1;
        END_IF;
    END_IF;

    // Event "Pumpcellars_HeadPumpcellar1_SensorTank_u_S2on".
    IF NOT progress THEN
        b1 := (state0.dvar_M_HPC1_HWSensorS2) = (elit_off);
        b1 := b1 AND (ivar_M_HPC1_HWSensorS2_ON);
        b1 := b1 AND ((state0.dvar_M_Pumpcellars_HeadPumpcellar1_SensorTank) = (elit_S1));
        IF b1 THEN
            progress := TRUE;
            state1 := state0;

            state1.dvar_M_HPC1_HWSensorS2 := elit_on;
            state1.dvar_M_Pumpcellars_HeadPumpcellar1_SensorTank := elit_S2;

            state0 := state1;
        END_IF;
    END_IF;

    // Event "Pumpcellars_HeadPumpcellar1_SensorTank_u_S3off".
    IF NOT progress THEN
        b1 := (state0.dvar_M_HPC1_HWSensorS3) = (elit_on);
        b1 := b1 AND (NOT(ivar_M_HPC1_HWSensorS3_ON));
        b1 := b1 AND ((state0.dvar_M_Pumpcellars_HeadPumpcellar1_SensorTank) = (elit_S3));
        IF b1 THEN
            b2 := (state0.dvar_M_Pumpcellars_HeadPumpcellar1_Pump1) = (elit_on);
            b2 := b2 OR ((state0.dvar_M_Pumpcellars_HeadPumpcellar1_Pump2) = (elit_on));
            b1 := b1 AND (b2);
        END_IF;
        IF b1 THEN
            progress := TRUE;
            state1 := state0;

            state1.dvar_M_HPC1_HWSensorS3 := elit_off;
            state1.dvar_M_Pumpcellars_HeadPumpcellar1_SensorTank := elit_S2;

            state0 := state1;
        END_IF;
    END_IF;

    // Event "Pumpcellars_HeadPumpcellar1_SensorTank_u_S3on".
    IF NOT progress THEN
        b1 := (state0.dvar_M_HPC1_HWSensorS3) = (elit_off);
        b1 := b1 AND (ivar_M_HPC1_HWSensorS3_ON);
        b1 := b1 AND ((state0.dvar_M_Pumpcellars_HeadPumpcellar1_SensorTank) = (elit_S2));
        IF b1 THEN
            progress := TRUE;
            state1 := state0;

            state1.dvar_M_HPC1_HWSensorS3 := elit_on;
            state1.dvar_M_Pumpcellars_HeadPumpcellar1_SensorTank := elit_S3;

            state0 := state1;
        END_IF;
    END_IF;

    // Event "Pumpcellars_HeadPumpcellar1_SensorTank_u_S4off".
    IF NOT progress THEN
        b1 := (state0.dvar_M_HPC1_HWSensorS4) = (elit_on);
        b1 := b1 AND (NOT(ivar_M_HPC1_HWSensorS4_ON));
        b1 := b1 AND ((state0.dvar_M_Pumpcellars_HeadPumpcellar1_SensorTank) = (elit_S4));
        IF b1 THEN
            b2 := (state0.dvar_M_Pumpcellars_HeadPumpcellar1_Pump1) = (elit_on);
            b2 := b2 OR ((state0.dvar_M_Pumpcellars_HeadPumpcellar1_Pump2) = (elit_on));
            b1 := b1 AND (b2);
        END_IF;
        IF b1 THEN
            progress := TRUE;
            state1 := state0;

            state1.dvar_M_HPC1_HWSensorS4 := elit_off;
            state1.dvar_M_Pumpcellars_HeadPumpcellar1_SensorTank := elit_S3;

            state0 := state1;
        END_IF;
    END_IF;

    // Event "Pumpcellars_HeadPumpcellar1_SensorTank_u_S4on".
    IF NOT progress THEN
        b1 := (state0.dvar_M_HPC1_HWSensorS4) = (elit_off);
        b1 := b1 AND (ivar_M_HPC1_HWSensorS4_ON);
        b1 := b1 AND ((state0.dvar_M_Pumpcellars_HeadPumpcellar1_SensorTank) = (elit_S3));
        IF b1 THEN
            progress := TRUE;
            state1 := state0;

            state1.dvar_M_HPC1_HWSensorS4 := elit_on;
            state1.dvar_M_Pumpcellars_HeadPumpcellar1_SensorTank := elit_S4;

            state0 := state1;
        END_IF;
    END_IF;

    // Event "Pumpcellars_HeadPumpcellar1_SensorTank_u_S5off".
    IF NOT progress THEN
        b1 := (state0.dvar_M_HPC1_HWSensorS5) = (elit_on);
        b1 := b1 AND (NOT(ivar_M_HPC1_HWSensorS5_ON));
        b1 := b1 AND ((state0.dvar_M_Pumpcellars_HeadPumpcellar1_SensorTank) = (elit_S5));
        IF b1 THEN
            b2 := (state0.dvar_M_Pumpcellars_HeadPumpcellar1_Pump1) = (elit_on);
            b2 := b2 OR ((state0.dvar_M_Pumpcellars_HeadPumpcellar1_Pump2) = (elit_on));
            b1 := b1 AND (b2);
        END_IF;
        IF b1 THEN
            progress := TRUE;
            state1 := state0;

            state1.dvar_M_HPC1_HWSensorS5 := elit_off;
            state1.dvar_M_Pumpcellars_HeadPumpcellar1_SensorTank := elit_S4;

            state0 := state1;
        END_IF;
    END_IF;

    // Event "Pumpcellars_HeadPumpcellar1_SensorTank_u_S5on".
    IF NOT progress THEN
        b1 := (state0.dvar_M_HPC1_HWSensorS5) = (elit_off);
        b1 := b1 AND (ivar_M_HPC1_HWSensorS5_ON);
        b1 := b1 AND ((state0.dvar_M_Pumpcellars_HeadPumpcellar1_SensorTank) = (elit_S4));
        IF b1 THEN
            progress := TRUE;
            state1 := state0;

            state1.dvar_M_HPC1_HWSensorS5 := elit_on;
            state1.dvar_M_Pumpcellars_HeadPumpcellar1_SensorTank := elit_S5;

            state0 := state1;
        END_IF;
    END_IF;

    // Event "Pumpcellars_MiddlePumpcellar_Control_ButtonAuto_u_push".
    IF NOT progress THEN
        b1 := (state0.dvar_M_HWMPCControlButtonAuto) = (elit_X);
        b1 := b1 AND (ivar_M_HWMPCControlButtonAuto_PUSHED);
        b1 := b1 AND (NOT(state0.dvar_M_HWMPCControlButtonAuto_StopLoop));
        b1 := b1 AND ((state0.dvar_M_Pumpcellars_MiddlePumpcellar_Control_ButtonAuto) = (elit_X));
        IF b1 THEN
            b3 := (state0.dvar_M_Pumpcellars_MiddlePumpcellar_Control_Observer) = (elit_unpressed);
            IF b3 THEN
                b4 := (state0.dvar_M_Pumpcellars_MiddlePumpcellar_Control_Mode) = (elit_manual);
                b4 := b4 OR ((state0.dvar_M_Pumpcellars_MiddlePumpcellar_Control_Mode) <> (elit_manual));
                b3 := b3 AND (b4);
            END_IF;
            b2 := b3;
            b2 := b2 OR ((state0.dvar_M_Pumpcellars_MiddlePumpcellar_Control_Observer) = (elit_autoPressed));
            b2 := b2 OR ((state0.dvar_M_Pumpcellars_MiddlePumpcellar_Control_Observer) = (elit_manualPressed));
            b2 := b2 OR ((state0.dvar_M_Pumpcellars_MiddlePumpcellar_Control_Observer) = (elit_storePressed));
            b2 := b2 OR ((state0.dvar_M_Pumpcellars_MiddlePumpcellar_Control_Observer) = (elit_drainPressed));
            b2 := b2 OR ((state0.dvar_M_Pumpcellars_MiddlePumpcellar_Control_Observer) = (elit_offPressed));
            b1 := b1 AND (b2);
        END_IF;
        IF b1 THEN
            progress := TRUE;
            state1 := state0;

            state1.dvar_M_HWMPCControlButtonAuto_StopLoop := TRUE;
            IF (((state0.dvar_M_Pumpcellars_MiddlePumpcellar_Control_Observer) = (elit_unpressed)) AND ((state0.dvar_M_Pumpcellars_MiddlePumpcellar_Control_Mode) = (elit_manual))) THEN
                state1.dvar_M_Pumpcellars_MiddlePumpcellar_Control_Observer := elit_autoPressed;
            ELSIF (((state0.dvar_M_Pumpcellars_MiddlePumpcellar_Control_Observer) = (elit_unpressed)) AND ((state0.dvar_M_Pumpcellars_MiddlePumpcellar_Control_Mode) <> (elit_manual))) THEN
                state1.dvar_M_Pumpcellars_MiddlePumpcellar_Control_Observer := elit_unpressed;
            ELSIF ((state0.dvar_M_Pumpcellars_MiddlePumpcellar_Control_Observer) = (elit_autoPressed)) THEN
                state1.dvar_M_Pumpcellars_MiddlePumpcellar_Control_Observer := elit_autoPressed;
            ELSIF ((state0.dvar_M_Pumpcellars_MiddlePumpcellar_Control_Observer) = (elit_manualPressed)) THEN
                state1.dvar_M_Pumpcellars_MiddlePumpcellar_Control_Observer := elit_manualPressed;
            ELSIF ((state0.dvar_M_Pumpcellars_MiddlePumpcellar_Control_Observer) = (elit_storePressed)) THEN
                state1.dvar_M_Pumpcellars_MiddlePumpcellar_Control_Observer := elit_storePressed;
            ELSIF ((state0.dvar_M_Pumpcellars_MiddlePumpcellar_Control_Observer) = (elit_drainPressed)) THEN
                state1.dvar_M_Pumpcellars_MiddlePumpcellar_Control_Observer := elit_drainPressed;
            ELSIF ((state0.dvar_M_Pumpcellars_MiddlePumpcellar_Control_Observer) = (elit_offPressed)) THEN
                state1.dvar_M_Pumpcellars_MiddlePumpcellar_Control_Observer := elit_offPressed;
            END_IF;

            state0 := state1;
        END_IF;
    END_IF;

    // Event "Pumpcellars_MiddlePumpcellar_Control_ButtonDrain_u_push".
    IF NOT progress THEN
        b1 := (state0.dvar_M_HWMPCModeButtonDrain) = (elit_X);
        b1 := b1 AND (ivar_M_HWMPCModeButtonDrain_PUSHED);
        b1 := b1 AND (NOT(state0.dvar_M_HWMPCModeButtonDrain_StopLoop));
        b1 := b1 AND ((state0.dvar_M_Pumpcellars_MiddlePumpcellar_Control_ButtonDrain) = (elit_X));
        IF b1 THEN
            b3 := (state0.dvar_M_Pumpcellars_MiddlePumpcellar_Control_Observer) = (elit_unpressed);
            IF b3 THEN
                b5 := (state0.dvar_M_Pumpcellars_MiddlePumpcellar_Control_Mode) = (elit_manual);
                b5 := b5 AND ((state0.dvar_M_Pumpcellars_MiddlePumpcellar_Mode) <> (elit_drain));
                b4 := b5;
                b4 := b4 OR (NOT(((state0.dvar_M_Pumpcellars_MiddlePumpcellar_Control_Mode) = (elit_manual)) AND ((state0.dvar_M_Pumpcellars_MiddlePumpcellar_Mode) <> (elit_drain))));
                b3 := b3 AND (b4);
            END_IF;
            b2 := b3;
            b2 := b2 OR ((state0.dvar_M_Pumpcellars_MiddlePumpcellar_Control_Observer) = (elit_autoPressed));
            b2 := b2 OR ((state0.dvar_M_Pumpcellars_MiddlePumpcellar_Control_Observer) = (elit_manualPressed));
            b2 := b2 OR ((state0.dvar_M_Pumpcellars_MiddlePumpcellar_Control_Observer) = (elit_storePressed));
            b2 := b2 OR ((state0.dvar_M_Pumpcellars_MiddlePumpcellar_Control_Observer) = (elit_drainPressed));
            b2 := b2 OR ((state0.dvar_M_Pumpcellars_MiddlePumpcellar_Control_Observer) = (elit_offPressed));
            b1 := b1 AND (b2);
        END_IF;
        IF b1 THEN
            progress := TRUE;
            state1 := state0;

            state1.dvar_M_HWMPCModeButtonDrain_StopLoop := TRUE;
            IF (((state0.dvar_M_Pumpcellars_MiddlePumpcellar_Control_Observer) = (elit_unpressed)) AND (((state0.dvar_M_Pumpcellars_MiddlePumpcellar_Control_Mode) = (elit_manual)) AND ((state0.dvar_M_Pumpcellars_MiddlePumpcellar_Mode) <> (elit_drain)))) THEN
                state1.dvar_M_Pumpcellars_MiddlePumpcellar_Control_Observer := elit_drainPressed;
            ELSIF (((state0.dvar_M_Pumpcellars_MiddlePumpcellar_Control_Observer) = (elit_unpressed)) AND (NOT(((state0.dvar_M_Pumpcellars_MiddlePumpcellar_Control_Mode) = (elit_manual)) AND ((state0.dvar_M_Pumpcellars_MiddlePumpcellar_Mode) <> (elit_drain))))) THEN
                state1.dvar_M_Pumpcellars_MiddlePumpcellar_Control_Observer := elit_unpressed;
            ELSIF ((state0.dvar_M_Pumpcellars_MiddlePumpcellar_Control_Observer) = (elit_autoPressed)) THEN
                state1.dvar_M_Pumpcellars_MiddlePumpcellar_Control_Observer := elit_autoPressed;
            ELSIF ((state0.dvar_M_Pumpcellars_MiddlePumpcellar_Control_Observer) = (elit_manualPressed)) THEN
                state1.dvar_M_Pumpcellars_MiddlePumpcellar_Control_Observer := elit_manualPressed;
            ELSIF ((state0.dvar_M_Pumpcellars_MiddlePumpcellar_Control_Observer) = (elit_storePressed)) THEN
                state1.dvar_M_Pumpcellars_MiddlePumpcellar_Control_Observer := elit_storePressed;
            ELSIF ((state0.dvar_M_Pumpcellars_MiddlePumpcellar_Control_Observer) = (elit_drainPressed)) THEN
                state1.dvar_M_Pumpcellars_MiddlePumpcellar_Control_Observer := elit_drainPressed;
            ELSIF ((state0.dvar_M_Pumpcellars_MiddlePumpcellar_Control_Observer) = (elit_offPressed)) THEN
                state1.dvar_M_Pumpcellars_MiddlePumpcellar_Control_Observer := elit_offPressed;
            END_IF;

            state0 := state1;
        END_IF;
    END_IF;

    // Event "Pumpcellars_MiddlePumpcellar_Control_ButtonManual_u_push".
    IF NOT progress THEN
        b1 := (state0.dvar_M_HWMPCControlButtonManual) = (elit_X);
        b1 := b1 AND (ivar_M_HWMPCControlButtonManual_PUSHED);
        b1 := b1 AND (NOT(state0.dvar_M_HWMPCControlButtonManual_StopLoop));
        b1 := b1 AND ((state0.dvar_M_Pumpcellars_MiddlePumpcellar_Control_ButtonManual) = (elit_X));
        IF b1 THEN
            b3 := (state0.dvar_M_Pumpcellars_MiddlePumpcellar_Control_Observer) = (elit_unpressed);
            IF b3 THEN
                b4 := (state0.dvar_M_Pumpcellars_MiddlePumpcellar_Control_Mode) = (elit_auto);
                b4 := b4 OR ((state0.dvar_M_Pumpcellars_MiddlePumpcellar_Control_Mode) <> (elit_auto));
                b3 := b3 AND (b4);
            END_IF;
            b2 := b3;
            b2 := b2 OR ((state0.dvar_M_Pumpcellars_MiddlePumpcellar_Control_Observer) = (elit_autoPressed));
            b2 := b2 OR ((state0.dvar_M_Pumpcellars_MiddlePumpcellar_Control_Observer) = (elit_manualPressed));
            b2 := b2 OR ((state0.dvar_M_Pumpcellars_MiddlePumpcellar_Control_Observer) = (elit_storePressed));
            b2 := b2 OR ((state0.dvar_M_Pumpcellars_MiddlePumpcellar_Control_Observer) = (elit_drainPressed));
            b2 := b2 OR ((state0.dvar_M_Pumpcellars_MiddlePumpcellar_Control_Observer) = (elit_offPressed));
            b1 := b1 AND (b2);
        END_IF;
        IF b1 THEN
            progress := TRUE;
            state1 := state0;

            state1.dvar_M_HWMPCControlButtonManual_StopLoop := TRUE;
            IF (((state0.dvar_M_Pumpcellars_MiddlePumpcellar_Control_Observer) = (elit_unpressed)) AND ((state0.dvar_M_Pumpcellars_MiddlePumpcellar_Control_Mode) = (elit_auto))) THEN
                state1.dvar_M_Pumpcellars_MiddlePumpcellar_Control_Observer := elit_manualPressed;
            ELSIF (((state0.dvar_M_Pumpcellars_MiddlePumpcellar_Control_Observer) = (elit_unpressed)) AND ((state0.dvar_M_Pumpcellars_MiddlePumpcellar_Control_Mode) <> (elit_auto))) THEN
                state1.dvar_M_Pumpcellars_MiddlePumpcellar_Control_Observer := elit_unpressed;
            ELSIF ((state0.dvar_M_Pumpcellars_MiddlePumpcellar_Control_Observer) = (elit_autoPressed)) THEN
                state1.dvar_M_Pumpcellars_MiddlePumpcellar_Control_Observer := elit_autoPressed;
            ELSIF ((state0.dvar_M_Pumpcellars_MiddlePumpcellar_Control_Observer) = (elit_manualPressed)) THEN
                state1.dvar_M_Pumpcellars_MiddlePumpcellar_Control_Observer := elit_manualPressed;
            ELSIF ((state0.dvar_M_Pumpcellars_MiddlePumpcellar_Control_Observer) = (elit_storePressed)) THEN
                state1.dvar_M_Pumpcellars_MiddlePumpcellar_Control_Observer := elit_storePressed;
            ELSIF ((state0.dvar_M_Pumpcellars_MiddlePumpcellar_Control_Observer) = (elit_drainPressed)) THEN
                state1.dvar_M_Pumpcellars_MiddlePumpcellar_Control_Observer := elit_drainPressed;
            ELSIF ((state0.dvar_M_Pumpcellars_MiddlePumpcellar_Control_Observer) = (elit_offPressed)) THEN
                state1.dvar_M_Pumpcellars_MiddlePumpcellar_Control_Observer := elit_offPressed;
            END_IF;

            state0 := state1;
        END_IF;
    END_IF;

    // Event "Pumpcellars_MiddlePumpcellar_Control_ButtonOff_u_push".
    IF NOT progress THEN
        b1 := (state0.dvar_M_HWMPCModeButtonOff) = (elit_X);
        b1 := b1 AND (ivar_M_HWMPCModeButtonOff_PUSHED);
        b1 := b1 AND (NOT(state0.dvar_M_HWMPCModeButtonOff_StopLoop));
        b1 := b1 AND ((state0.dvar_M_Pumpcellars_MiddlePumpcellar_Control_ButtonOff) = (elit_X));
        IF b1 THEN
            b3 := (state0.dvar_M_Pumpcellars_MiddlePumpcellar_Control_Observer) = (elit_unpressed);
            IF b3 THEN
                b5 := (state0.dvar_M_Pumpcellars_MiddlePumpcellar_Control_Mode) = (elit_manual);
                b5 := b5 AND ((state0.dvar_M_Pumpcellars_MiddlePumpcellar_Mode) <> (elit_off));
                b4 := b5;
                b4 := b4 OR (NOT(((state0.dvar_M_Pumpcellars_MiddlePumpcellar_Control_Mode) = (elit_manual)) AND ((state0.dvar_M_Pumpcellars_MiddlePumpcellar_Mode) <> (elit_off))));
                b3 := b3 AND (b4);
            END_IF;
            b2 := b3;
            b2 := b2 OR ((state0.dvar_M_Pumpcellars_MiddlePumpcellar_Control_Observer) = (elit_autoPressed));
            b2 := b2 OR ((state0.dvar_M_Pumpcellars_MiddlePumpcellar_Control_Observer) = (elit_manualPressed));
            b2 := b2 OR ((state0.dvar_M_Pumpcellars_MiddlePumpcellar_Control_Observer) = (elit_storePressed));
            b2 := b2 OR ((state0.dvar_M_Pumpcellars_MiddlePumpcellar_Control_Observer) = (elit_drainPressed));
            b2 := b2 OR ((state0.dvar_M_Pumpcellars_MiddlePumpcellar_Control_Observer) = (elit_offPressed));
            b1 := b1 AND (b2);
        END_IF;
        IF b1 THEN
            progress := TRUE;
            state1 := state0;

            state1.dvar_M_HWMPCModeButtonOff_StopLoop := TRUE;
            IF (((state0.dvar_M_Pumpcellars_MiddlePumpcellar_Control_Observer) = (elit_unpressed)) AND (((state0.dvar_M_Pumpcellars_MiddlePumpcellar_Control_Mode) = (elit_manual)) AND ((state0.dvar_M_Pumpcellars_MiddlePumpcellar_Mode) <> (elit_off)))) THEN
                state1.dvar_M_Pumpcellars_MiddlePumpcellar_Control_Observer := elit_offPressed;
            ELSIF (((state0.dvar_M_Pumpcellars_MiddlePumpcellar_Control_Observer) = (elit_unpressed)) AND (NOT(((state0.dvar_M_Pumpcellars_MiddlePumpcellar_Control_Mode) = (elit_manual)) AND ((state0.dvar_M_Pumpcellars_MiddlePumpcellar_Mode) <> (elit_off))))) THEN
                state1.dvar_M_Pumpcellars_MiddlePumpcellar_Control_Observer := elit_unpressed;
            ELSIF ((state0.dvar_M_Pumpcellars_MiddlePumpcellar_Control_Observer) = (elit_autoPressed)) THEN
                state1.dvar_M_Pumpcellars_MiddlePumpcellar_Control_Observer := elit_autoPressed;
            ELSIF ((state0.dvar_M_Pumpcellars_MiddlePumpcellar_Control_Observer) = (elit_manualPressed)) THEN
                state1.dvar_M_Pumpcellars_MiddlePumpcellar_Control_Observer := elit_manualPressed;
            ELSIF ((state0.dvar_M_Pumpcellars_MiddlePumpcellar_Control_Observer) = (elit_storePressed)) THEN
                state1.dvar_M_Pumpcellars_MiddlePumpcellar_Control_Observer := elit_storePressed;
            ELSIF ((state0.dvar_M_Pumpcellars_MiddlePumpcellar_Control_Observer) = (elit_drainPressed)) THEN
                state1.dvar_M_Pumpcellars_MiddlePumpcellar_Control_Observer := elit_drainPressed;
            ELSIF ((state0.dvar_M_Pumpcellars_MiddlePumpcellar_Control_Observer) = (elit_offPressed)) THEN
                state1.dvar_M_Pumpcellars_MiddlePumpcellar_Control_Observer := elit_offPressed;
            END_IF;

            state0 := state1;
        END_IF;
    END_IF;

    // Event "Pumpcellars_MiddlePumpcellar_Control_ButtonStore_u_push".
    IF NOT progress THEN
        b1 := (state0.dvar_M_HWMPCModeButtonStore) = (elit_X);
        b1 := b1 AND (ivar_M_HWMPCModeButtonStore_PUSHED);
        b1 := b1 AND (NOT(state0.dvar_M_HWMPCModeButtonStore_StopLoop));
        b1 := b1 AND ((state0.dvar_M_Pumpcellars_MiddlePumpcellar_Control_ButtonStore) = (elit_X));
        IF b1 THEN
            b3 := (state0.dvar_M_Pumpcellars_MiddlePumpcellar_Control_Observer) = (elit_unpressed);
            IF b3 THEN
                b5 := (state0.dvar_M_Pumpcellars_MiddlePumpcellar_Control_Mode) = (elit_manual);
                b5 := b5 AND ((state0.dvar_M_Pumpcellars_MiddlePumpcellar_Mode) <> (elit_store));
                b4 := b5;
                b4 := b4 OR (NOT(((state0.dvar_M_Pumpcellars_MiddlePumpcellar_Control_Mode) = (elit_manual)) AND ((state0.dvar_M_Pumpcellars_MiddlePumpcellar_Mode) <> (elit_store))));
                b3 := b3 AND (b4);
            END_IF;
            b2 := b3;
            b2 := b2 OR ((state0.dvar_M_Pumpcellars_MiddlePumpcellar_Control_Observer) = (elit_autoPressed));
            b2 := b2 OR ((state0.dvar_M_Pumpcellars_MiddlePumpcellar_Control_Observer) = (elit_manualPressed));
            b2 := b2 OR ((state0.dvar_M_Pumpcellars_MiddlePumpcellar_Control_Observer) = (elit_storePressed));
            b2 := b2 OR ((state0.dvar_M_Pumpcellars_MiddlePumpcellar_Control_Observer) = (elit_drainPressed));
            b2 := b2 OR ((state0.dvar_M_Pumpcellars_MiddlePumpcellar_Control_Observer) = (elit_offPressed));
            b1 := b1 AND (b2);
        END_IF;
        IF b1 THEN
            progress := TRUE;
            state1 := state0;

            state1.dvar_M_HWMPCModeButtonStore_StopLoop := TRUE;
            IF (((state0.dvar_M_Pumpcellars_MiddlePumpcellar_Control_Observer) = (elit_unpressed)) AND (((state0.dvar_M_Pumpcellars_MiddlePumpcellar_Control_Mode) = (elit_manual)) AND ((state0.dvar_M_Pumpcellars_MiddlePumpcellar_Mode) <> (elit_store)))) THEN
                state1.dvar_M_Pumpcellars_MiddlePumpcellar_Control_Observer := elit_storePressed;
            ELSIF (((state0.dvar_M_Pumpcellars_MiddlePumpcellar_Control_Observer) = (elit_unpressed)) AND (NOT(((state0.dvar_M_Pumpcellars_MiddlePumpcellar_Control_Mode) = (elit_manual)) AND ((state0.dvar_M_Pumpcellars_MiddlePumpcellar_Mode) <> (elit_store))))) THEN
                state1.dvar_M_Pumpcellars_MiddlePumpcellar_Control_Observer := elit_unpressed;
            ELSIF ((state0.dvar_M_Pumpcellars_MiddlePumpcellar_Control_Observer) = (elit_autoPressed)) THEN
                state1.dvar_M_Pumpcellars_MiddlePumpcellar_Control_Observer := elit_autoPressed;
            ELSIF ((state0.dvar_M_Pumpcellars_MiddlePumpcellar_Control_Observer) = (elit_manualPressed)) THEN
                state1.dvar_M_Pumpcellars_MiddlePumpcellar_Control_Observer := elit_manualPressed;
            ELSIF ((state0.dvar_M_Pumpcellars_MiddlePumpcellar_Control_Observer) = (elit_storePressed)) THEN
                state1.dvar_M_Pumpcellars_MiddlePumpcellar_Control_Observer := elit_storePressed;
            ELSIF ((state0.dvar_M_Pumpcellars_MiddlePumpcellar_Control_Observer) = (elit_drainPressed)) THEN
                state1.dvar_M_Pumpcellars_MiddlePumpcellar_Control_Observer := elit_drainPressed;
            ELSIF ((state0.dvar_M_Pumpcellars_MiddlePumpcellar_Control_Observer) = (elit_offPressed)) THEN
                state1.dvar_M_Pumpcellars_MiddlePumpcellar_Control_Observer := elit_offPressed;
            END_IF;

            state0 := state1;
        END_IF;
    END_IF;

    // Event "Pumpcellars_MiddlePumpcellar_Control_Mode_c_auto".
    IF NOT progress THEN
        b1 := (state0.dvar_M_HWMPCControlMode) = (elit_X);
        b1 := b1 AND ((state0.dvar_M_Pumpcellars_MiddlePumpcellar_Control_Mode) = (elit_manual));
        b1 := b1 AND ((state0.dvar_M_RequirementStateEvtExcls) = (elit_X));
        b1 := b1 AND ((state0.dvar_M_Pumpcellars_MiddlePumpcellar_Control_Observer) = (elit_autoPressed));
        b1 := b1 AND ((state0.dvar_M_sup1a) = (elit_X));
        b1 := b1 AND ((state0.dvar_M_sup2) = (elit_X));
        b1 := b1 AND ((state0.dvar_M_sup4) = (elit_X));
        IF b1 THEN
            progress := TRUE;
            state1 := state0;

            state1.dvar_M_HWMPCControlMode_AUTO := TRUE;
            state1.dvar_M_Pumpcellars_MiddlePumpcellar_Control_Mode := elit_auto;

            state0 := state1;
        END_IF;
    END_IF;

    // Event "Pumpcellars_MiddlePumpcellar_Control_Mode_c_manual".
    IF NOT progress THEN
        b1 := (state0.dvar_M_HWMPCControlMode) = (elit_X);
        b1 := b1 AND ((state0.dvar_M_Pumpcellars_MiddlePumpcellar_Control_Mode) = (elit_auto));
        b1 := b1 AND ((state0.dvar_M_RequirementStateEvtExcls) = (elit_X));
        b1 := b1 AND ((state0.dvar_M_Pumpcellars_MiddlePumpcellar_Control_Observer) = (elit_manualPressed));
        b1 := b1 AND ((state0.dvar_M_sup1a) = (elit_X));
        b1 := b1 AND ((state0.dvar_M_sup2) = (elit_X));
        b1 := b1 AND ((state0.dvar_M_sup4) = (elit_X));
        IF b1 THEN
            progress := TRUE;
            state1 := state0;

            state1.dvar_M_HWMPCControlMode_AUTO := FALSE;
            state1.dvar_M_Pumpcellars_MiddlePumpcellar_Control_Mode := elit_manual;

            state0 := state1;
        END_IF;
    END_IF;

    // Event "Pumpcellars_MiddlePumpcellar_Control_Observer_c_done".
    IF NOT progress THEN
        b1 := (state0.dvar_M_HWMPCControlButtonAuto) = (elit_X);
        b1 := b1 AND ((state0.dvar_M_HWMPCControlButtonManual) = (elit_X));
        b1 := b1 AND ((state0.dvar_M_HWMPCModeButtonDrain) = (elit_X));
        b1 := b1 AND ((state0.dvar_M_HWMPCModeButtonOff) = (elit_X));
        b1 := b1 AND ((state0.dvar_M_HWMPCModeButtonStore) = (elit_X));
        IF b1 THEN
            b3 := (state0.dvar_M_Pumpcellars_MiddlePumpcellar_Control_Observer) = (elit_autoPressed);
            b3 := b3 AND ((state0.dvar_M_Pumpcellars_MiddlePumpcellar_Control_Mode) = (elit_auto));
            b2 := b3;
            IF NOT(b2) THEN
                b3 := (state0.dvar_M_Pumpcellars_MiddlePumpcellar_Control_Observer) = (elit_manualPressed);
                b3 := b3 AND ((state0.dvar_M_Pumpcellars_MiddlePumpcellar_Control_Mode) = (elit_manual));
                b2 := b2 OR (b3);
            END_IF;
            IF NOT(b2) THEN
                b3 := (state0.dvar_M_Pumpcellars_MiddlePumpcellar_Control_Observer) = (elit_storePressed);
                b3 := b3 AND ((state0.dvar_M_Pumpcellars_MiddlePumpcellar_Mode) = (elit_store));
                b2 := b2 OR (b3);
            END_IF;
            IF NOT(b2) THEN
                b3 := (state0.dvar_M_Pumpcellars_MiddlePumpcellar_Control_Observer) = (elit_drainPressed);
                b3 := b3 AND ((state0.dvar_M_Pumpcellars_MiddlePumpcellar_Mode) = (elit_drain));
                b2 := b2 OR (b3);
            END_IF;
            IF NOT(b2) THEN
                b3 := (state0.dvar_M_Pumpcellars_MiddlePumpcellar_Control_Observer) = (elit_offPressed);
                b3 := b3 AND ((state0.dvar_M_Pumpcellars_MiddlePumpcellar_Mode) = (elit_off));
                b2 := b2 OR (b3);
            END_IF;
            b1 := b1 AND (b2);
        END_IF;
        b1 := b1 AND ((state0.dvar_M_sup1a) = (elit_X));
        b1 := b1 AND ((state0.dvar_M_sup2) = (elit_X));
        b1 := b1 AND ((state0.dvar_M_sup4) = (elit_X));
        IF b1 THEN
            progress := TRUE;
            state1 := state0;

            state1.dvar_M_HWMPCControlButtonAuto_StopLoop := FALSE;
            state1.dvar_M_HWMPCControlButtonManual_StopLoop := FALSE;
            state1.dvar_M_HWMPCModeButtonDrain_StopLoop := FALSE;
            state1.dvar_M_HWMPCModeButtonOff_StopLoop := FALSE;
            state1.dvar_M_HWMPCModeButtonStore_StopLoop := FALSE;
            IF (((state0.dvar_M_Pumpcellars_MiddlePumpcellar_Control_Observer) = (elit_autoPressed)) AND ((state0.dvar_M_Pumpcellars_MiddlePumpcellar_Control_Mode) = (elit_auto))) THEN
                state1.dvar_M_Pumpcellars_MiddlePumpcellar_Control_Observer := elit_unpressed;
            ELSIF (((state0.dvar_M_Pumpcellars_MiddlePumpcellar_Control_Observer) = (elit_manualPressed)) AND ((state0.dvar_M_Pumpcellars_MiddlePumpcellar_Control_Mode) = (elit_manual))) THEN
                state1.dvar_M_Pumpcellars_MiddlePumpcellar_Control_Observer := elit_unpressed;
            ELSIF (((state0.dvar_M_Pumpcellars_MiddlePumpcellar_Control_Observer) = (elit_storePressed)) AND ((state0.dvar_M_Pumpcellars_MiddlePumpcellar_Mode) = (elit_store))) THEN
                state1.dvar_M_Pumpcellars_MiddlePumpcellar_Control_Observer := elit_unpressed;
            ELSIF (((state0.dvar_M_Pumpcellars_MiddlePumpcellar_Control_Observer) = (elit_drainPressed)) AND ((state0.dvar_M_Pumpcellars_MiddlePumpcellar_Mode) = (elit_drain))) THEN
                state1.dvar_M_Pumpcellars_MiddlePumpcellar_Control_Observer := elit_unpressed;
            ELSIF (((state0.dvar_M_Pumpcellars_MiddlePumpcellar_Control_Observer) = (elit_offPressed)) AND ((state0.dvar_M_Pumpcellars_MiddlePumpcellar_Mode) = (elit_off))) THEN
                state1.dvar_M_Pumpcellars_MiddlePumpcellar_Control_Observer := elit_unpressed;
            END_IF;

            state0 := state1;
        END_IF;
    END_IF;

    // Event "Pumpcellars_MiddlePumpcellar_Mode_c_drain".
    IF NOT progress THEN
        b2 := (state0.dvar_M_Pumpcellars_MiddlePumpcellar_Mode) = (elit_store);
        b2 := b2 OR ((state0.dvar_M_Pumpcellars_MiddlePumpcellar_Mode) = (elit_off));
        b1 := b2;
        b1 := b1 AND ((state0.dvar_M_RequirementStateEvtExcls) = (elit_X));
        IF b1 THEN
            b2 := (state0.dvar_M_Pumpcellars_MiddlePumpcellar_Control_Observer) = (elit_unpressed);
            IF NOT(b2) THEN
                b3 := (state0.dvar_M_Pumpcellars_MiddlePumpcellar_Control_Mode) = (elit_manual);
                b3 := b3 AND ((state0.dvar_M_Pumpcellars_MiddlePumpcellar_Control_Observer) <> (elit_autoPressed));
                b2 := b2 OR (b3);
            END_IF;
            b1 := b1 AND (b2);
        END_IF;
        IF b1 THEN
            b3 := (state0.dvar_M_Pumpcellars_MiddlePumpcellar_Control_Mode) = (elit_auto);
            b3 := b3 AND ((state0.dvar_M_Pumpcellars_Traffictube1_ModeTraffictube_Observer) = (elit_operational));
            b3 := b3 AND ((state0.dvar_M_Pumpcellars_Traffictube2_ModeTraffictube_Observer) = (elit_operational));
            b2 := b3;
            IF NOT(b2) THEN
                b3 := (state0.dvar_M_Pumpcellars_MiddlePumpcellar_Control_Mode) = (elit_manual);
                b3 := b3 AND ((state0.dvar_M_Pumpcellars_MiddlePumpcellar_Control_Observer) = (elit_drainPressed));
                b2 := b2 OR (b3);
            END_IF;
            b1 := b1 AND (b2);
        END_IF;
        b1 := b1 AND ((state0.dvar_M_Mutex1Home_TokenTracker) = (elit_Home));
        b1 := b1 AND ((state0.dvar_M_Mutex2Home_TokenTracker) = (elit_Home));
        b1 := b1 AND ((state0.dvar_M_sup1a) = (elit_X));
        b1 := b1 AND ((state0.dvar_M_sup2) = (elit_X));
        b1 := b1 AND ((state0.dvar_M_sup4) = (elit_X));
        IF b1 THEN
            progress := TRUE;
            state1 := state0;

            IF ((state0.dvar_M_HWMPCMode) = (elit_drain)) THEN
                state1.dvar_M_HWMPCMode := elit_drain;
            ELSIF ((state0.dvar_M_HWMPCMode) = (elit_store)) THEN
                state1.dvar_M_HWMPCMode_DRAIN := TRUE;
                state1.dvar_M_HWMPCMode_STORE := FALSE;
                state1.dvar_M_HWMPCMode_OFF := FALSE;
                state1.dvar_M_HWMPCMode := elit_drain;
            ELSIF ((state0.dvar_M_HWMPCMode) = (elit_off)) THEN
                state1.dvar_M_HWMPCMode_DRAIN := TRUE;
                state1.dvar_M_HWMPCMode_STORE := FALSE;
                state1.dvar_M_HWMPCMode_OFF := FALSE;
                state1.dvar_M_HWMPCMode := elit_drain;
            END_IF;
            IF ((state0.dvar_M_Pumpcellars_MiddlePumpcellar_Mode) = (elit_store)) THEN
                state1.dvar_M_Pumpcellars_MiddlePumpcellar_Mode := elit_drain;
            ELSIF ((state0.dvar_M_Pumpcellars_MiddlePumpcellar_Mode) = (elit_off)) THEN
                state1.dvar_M_Pumpcellars_MiddlePumpcellar_Mode := elit_drain;
            END_IF;

            state0 := state1;
        END_IF;
    END_IF;

